// TwinCAT 3 PLC project Clara_20230419
// ProgramVersion: 3.1.4022.7
// CompilerDefines: VISU_USEWSTRING
// libraries:
//   CAA Memory, * (CAA Technical Workgroup)
//   CmpBitmapPool, * (System)
//   Tc2_EtherCAT, * (Beckhoff Automation GmbH)
//   Tc2_IoFunctions, * (Beckhoff Automation GmbH)
//   Tc2_MC2, * (Beckhoff Automation GmbH)
//   Tc2_MDP, * (Beckhoff Automation GmbH)
//   Tc2_ModbusRTU, * (Beckhoff Automation GmbH)
//   Tc2_SerialCom, * (Beckhoff Automation GmbH)
//   Tc2_Standard, * (Beckhoff Automation GmbH)
//   Tc2_SUPS, * (Beckhoff Automation GmbH)
//   Tc2_System, * (Beckhoff Automation GmbH)
//   Tc2_SystemCX, * (Beckhoff Automation GmbH)
//   Tc2_Utilities, * (Beckhoff Automation GmbH)
//   Tc3_Module, * (Beckhoff Automation GmbH)
//   VisuDialogs, * (System)
//   VisuSymbols,3.5.10.0,System
// project tree:
//   DUTs/01_ST_IO/ ST_Input.TcDUT, ST_IO_FootPedal.TcDUT, ST_Output.TcDUT (not stored)
//   DUTs/02_PLC/ stAxis.TcDUT, stFootPedal.TcDUT (not stored), stISS.TcDUT, stSubTank.TcDUT, stMaintenanceUnit.TcDUT (not stored), stRollToRoll.TcDUT (not stored), stRtu.TcDUT, stSafetyGuard.TcDUT (not stored), stSpitUnit.TcDUT, stSystemEnvironment.TcDUT (not stored), stTableVacuum.TcDUT, stUpDownSlot.TcDUT (not stored), stUVLed.TcDUT
//   Enum_Text/Enum/PLC/ AxisStateEnum.TcDUT, Axis_XY_ErrorEnum.TcDUT, Axis_Z_ErrorEnum.TcDUT (not stored), EnvironmentErrorEnum.TcDUT (not stored), EnvironmentStateEnum.TcDUT (not stored), FootPedalErrorEnum.TcDUT, FootPedalStateEnum.TcDUT, ISSErrorEnum.TcDUT, SubTankErrorEnum.TcDUT (not stored), ISSStateEnum.TcDUT (not stored), SubTankInkEnum.TcDUT, SubTankStateEnum.TcDUT, MUErrorEnum.TcDUT, MUStateEnum.TcDUT, RTRErrorEnum.TcDUT (not stored), RTRStateEnum.TcDUT (not stored), SafetyGuardErrorEnum.TcDUT (not stored), SafetyGuardStateEnum.TcDUT (not stored), SpitUnitErrorEnum.TcDUT (not stored), SpitUnitStateEnum.TcDUT (not stored), SwapInfoEnum.TcDUT, TabVacErrorEnum.TcDUT (not stored), TabVacStateEnum.TcDUT, UpDownSlotErrorEnum.TcDUT (not stored), UpDownSlotStateEnum.TcDUT (not stored), UVLedErrorEnum.TcDUT (not stored), UVLedStateEnum.TcDUT (not stored)
//   Enum_Text/Enum/TwinSafe/ TwinSAFE_FB_ESTOP_State_Enum.TcDUT, TwinSAFE_Group_State_Enum.TcDUT (not stored)
//   Global Variables/ _01_Global_Variables.TcGVL, _04_Global_Variables_InOutput.TcGVL
//   / GlobalTextList.TcGTLO, ImagePool.TcIPO (not stored), PlcTask.TcTTO, Task_com.TcTTO, 视图管理器.TcVMO (not stored)
//   GVLs/ COMM.TcGVL, GVL.TcGVL, GVL_Alarm.TcGVL, GVL_API.TcGVL (not stored)
//   POUs/000_程序辅助系统/报警/Data types/ Alm_AlarmHistoryType.TcDUT (not stored), Alm_AlarmType.TcDUT, Alm_AlmMsg.TcDUT, Alm_EventClass.TcDUT
//   POUs/000_程序辅助系统/报警/diag_FB/ ethercatinfo_read.TcPOU (not stored)
//   POUs/000_程序辅助系统/报警/Alarm_FB/ FB_AlarmMain.TcPOU, FB_DiagDataLogging_S.TcPOU (not stored), FB_SetAlarm.TcPOU (not stored), SW_FormatWstring.TcPOU
//   POUs/000_程序辅助系统/报警/Alarm_FB/Products/ FB_DirectoryCopy.TcPOU (not stored), FB_FileCopy.TcPOU
//   POUs/000_程序辅助系统/报警/ MAIN_Alarm.TcPOU (not stored)
//   POUs/000_程序辅助系统/系统功能/ P_UPS.TcPOU (not stored), systime.TcPOU
//   POUs/001_FB/ FB_Buzzer.TcPOU, FB_count.TcPOU (not stored), FB_SQUARE.TcPOU, FB_WriteAnalog.TcPOU (not stored)
//   POUs/002_Modbus/BackPrg/ PRG_COMM.TcPOU
//   POUs/002_Modbus/ PRG_SerialComm.TcPOU (not stored), P_Modbus.TcPOU, P_Modbus_RTU.TcPOU (not stored)
//   POUs/003_Input_Output/ IO_Link.TcPOU, P_API_IO.TcPOU (not stored)
//   POUs/010_Motion/MotionBase/ FB_Home_Z.TcPOU (not stored), FB_Home_X.TcPOU, FB_MoveFS_Exte.TcPOU, FB_MoveSS_Exte.TcPOU, FB_MoveZ_Exte.TcPOU
//   POUs/010_Motion/XMove/ P_FastScan.TcPOU
//   POUs/010_Motion/YMove/ P_SlowScan.TcPOU
//   POUs/010_Motion/ZMove/ P_Z_Axis.TcPOU
//   POUs/030_MediaTransport/TableVacuum/FB/ FB_TableVacuum.TcPOU (not stored)
//   POUs/030_MediaTransport/UpDownSlot/FB/ FB_UpDownSlotS1.TcPOU, FB_UpDownSlotS2_S6.TcPOU
//   POUs/040_System/FootPedal/FB/ FB_FootPedal.TcPOU
//   POUs/040_System/SafetyGuard/FB/ FB_SafetyGuard.TcPOU (not stored)
//   POUs/040_System/SafetyGuard/ P_SafetyGuard.TcPOU (not stored)
//   POUs/040_System/SystemEnvironment/FB/ FB_SystemEnvironment.TcPOU
//   POUs/050_InkSystem/ISS/ P_ISS.TcPOU
//   POUs/050_InkSystem/ P_InkSystem.TcPOU (not stored)
//   POUs/050_InkSystem/搅拌_吸废墨/FB/ FB_Stirrer.TcPOU (not stored)
//   POUs/050_InkSystem/搅拌_吸废墨/ P_Stirrer_WastePump.TcPOU (not stored)
//   POUs/030_MediaTransport/ P_MediaTransport.TcPOU
//   POUs/030_MediaTransport/TableVacuum/ P_TableVacuum.TcPOU (not stored)
//   POUs/030_MediaTransport/UpDownSlot/ P_UpDownSlot.TcPOU (not stored)
//   POUs/010_Motion/MotionBase/PTP/ Axis_IO.TcPOU, Axis_PTP_CoE.TcPOU (not stored)
//   POUs/010_Motion/ P_Motion.TcPOU (not stored)
//   POUs/060_UVLed/FB/ FB_UVLed_L.TcPOU (not stored), FB_UVLed_R.TcPOU (not stored)
//   POUs/070_RollToRoll/FB/ FB_RollToRoll_Torque.TcPOU
//   POUs/100_SubTank/FB/ FB_Circulation.TcPOU, FB_SubTank_C.TcPOU, FB_SubTank_W.TcPOU
//   POUs/100_SubTank/ P_SubTank.TcPOU
//   POUs/999_TwinSAFE/ P_TwinSAFE.TcPOU
//   POUs/ MAIN.TcPOU (not stored)
//   POUs/070_RollToRoll/ P_RollToRoll.TcPOU (not stored)
//   POUs/040_System/FootPedal/ P_FootPedal.TcPOU (not stored)
//   POUs/040_System/ P_System.TcPOU (not stored)
//   POUs/040_System/SystemEnvironment/ P_SystemEnvironment.TcPOU
//   POUs/060_UVLed/ P_UVLed.TcPOU (not stored)
//   POUs/090MaintenanceUnit/FB/ FB_Auto_Cycles_Swap.TcPOU (not stored), FB_drip_purge.TcPOU
//   POUs/090MaintenanceUnit/ P_MaintenanceUnit.TcPOU (not stored)
//   POUs/080SpitUnit/FB/ FB_HomeSpitUnit.TcPOU, FB_MoveSpitUnit_Exte.TcPOU
//   POUs/080SpitUnit/ P_SpitUnit.TcPOU
//   VISUs/base/ title.TcVIS
//   VISUs/Components/IO_Components/ F99_IO_IO.TcVIS, F99_IO_IO_1.TcVIS, F99_IO_IO_2.TcVIS
//   VISUs/Components/ VIS_FootPedal.TcVIS (not stored), VIS_Drip_purge.TcVIS (not stored), VIS_SubTank.TcVIS, VIS_SystemEnvironment.TcVIS (not stored), VIS_ISS.TcVIS (not stored), VIS_MU.TcVIS (not stored), VIS_RTR_1.TcVIS (not stored), VIS_RTR_2.TcVIS, VIS_SaftyGuard.TcVIS (not stored), VIS_SpitUnit.TcVIS, VIS_TabVac.TcVIS, VIS_UpDownSlot.TcVIS
//   VISUs/HMI_IO监控文字/ EL1809_M_1.TcTLO, EL1809_M_2.TcTLO, EL1809_M_3.TcTLO, EL1809_S_1.TcTLO, EL1809_S_2.TcTLO (not stored), EL1904_M_1.TcTLO, EL1904_M_2.TcTLO, EL1904_M_3.TcTLO (not stored), EL1904_M_4.TcTLO (not stored), EL1904_M_5.TcTLO (not stored), EL2809_M_1.TcTLO (not stored), EL2809_M_2.TcTLO (not stored), EL2809_M_3.TcTLO (not stored), EL2809_M_4.TcTLO, EL2809_S_1.TcTLO (not stored), EL2904_M_1.TcTLO (not stored)
//   VISUs/ F99_Monitor.TcVIS (not stored), F7_RTR.TcVIS, F4_System.TcVIS (not stored), F1_AXIS.TcVIS, F5_InkSystem.TcVIS, F3_MediaTransport.TcVIS (not stored), F6_UVLed.TcVIS (not stored)
//   VISUs/VIS文本/PLC/ ISS_Object.TcTLO, subinklevel.TcTLO (not stored), TextListSpitUnitErrorid.TcTLO (not stored), TextListSpitUnitState.TcTLO, TextList_EnvironmentError.TcTLO, TextList_EnvironmentState.TcTLO, TextList_FootPedalerroid.TcTLO (not stored), TextList_SubTankerroid.TcTLO, TextList_FootPedalstate.TcTLO, TextList_ISSerrorid.TcTLO, TextList_ISSstate.TcTLO, TextList_MU_errorid.TcTLO, TextList_MU_state.TcTLO, TextList_RTRstate.TcTLO (not stored), TextList_RTR_errorid.TcTLO, TextList_SafetyGuarderrorid.TcTLO (not stored), TextList_SafetyGuardstate.TcTLO, TextList_SubTank_circuit.TcTLO, TextList_SwapInfo.TcTLO, TextList_tabvac_errorid.TcTLO, TextList_tabvac_state.TcTLO, TextList_UpDownSlot_errorid.TcTLO, TextList_UpDownSlot_state.TcTLO, TextList_UVLed_errorid.TcTLO (not stored), TextList_UVLed_state.TcTLO (not stored), TextList_xyErrorid.TcTLO, TextList_xyzState.TcTLO, TextList_zErrorid.TcTLO (not stored)
//   VISUs/VIS文本/TwinSafe/ TextList_TwinSAFE_FB_ESTOP_State.TcTLO, TextList_TwinSAFE_Group_State.TcTLO
//   VISUs/报警/ Visualization_ActEvent.TcVIS, Visualization_LogEvent.TcVIS (not stored), vis_arm.TcVIS
// real-time tasks:
//   TASK PlcTask: cycle T#10ms, priority 12, ADS port 350
//   TASK Task_com: cycle T#2ms, priority 6, ADS port 352
// motion (NC):
//   TASK NC-Task 1 SAF: cycle T#2ms, priority 4, ADS port 501
//   TASK NC-Task 1 SVB: cycle T#5ms, priority 10, ADS port 511
//   AXIS Axis_FS (id 1)
//     Dynamic: Acceleration=5927.27, Deceleration=5927.27, Jerk=27883
//     Velo: RefSearch=10, RefSync=10, SlowManual=50, FastManual=100
//     TargetPosControl: Time=0.005
//     OtherSettings: AllowMotionCmdToSlave=true
//     encoder EncType=19
//       EncPara: ScaleFactorNumerator=0.001, MaxCount=#xffffffff
//         Inc: RefSearchInverse=true, RefSyncInverse=false
//     drive DrvType=16
//       DrvPara: MaxCount=#xffffffff, DriveControlDWord=#x00020000
//         Analog: VeloReferenz=2000, TorqueSetpointScale=10, ScaleFactorActTorque=0.1
//         TimeComp: TaskDelayCycles=1
//     controller CtrType=1
//       CtrPara: PriorControlFactor=1
//         PosDiffControl: Range=250
//         Observer: BandWidth=20
//   AXIS Axis_SS (id 2)
//     Dynamic: Acceleration=274.92, Deceleration=274.92, Jerk=748.92
//     Velo: Maximum=174
//     OtherSettings: AllowMotionCmdToSlave=true
//     encoder EncType=19
//       EncPara: ScaleFactorNumerator=3.12605035e-07, Inverse=true, MaxCount=#xffffffff
//     drive DrvType=16
//       DrvPara: Inverse=true, MaxCount=#xffffffff, DriveControlDWord=#x00020000
//         Analog: VeloReferenz=180, TorqueSetpointScale=10, ScaleFactorActTorque=0.1
//         TimeComp: TaskDelayCycles=1
//     controller CtrType=1
//       CtrPara: PriorControlFactor=1
//         PosDiffControl: Range=50
//         Observer: BandWidth=20
//   AXIS Z_Axis (id 3)
//     Dynamic: Acceleration=33.4286, Deceleration=33.4286, Jerk=133.032
//     Velo: RefSearch=2, RefSync=2, SlowManual=8, FastManual=10, Maximum=15
//     OtherSettings: AllowMotionCmdToSlave=true
//     encoder EncType=19
//       EncPara: ScaleFactorNumerator=1.7881393e-08, MaxCount=#xffffffff
//         Inc: RefSearchInverse=true, RefSyncInverse=false
//     drive DrvType=16
//       DrvPara: MaxCount=#xffffffff, DriveControlDWord=#x00020000
//         Analog: VeloReferenz=15, TorqueSetpointScale=10, ScaleFactorActTorque=0.1
//         TimeComp: TaskDelayCycles=1
//     controller CtrType=1
//       CtrPara: PriorControlFactor=1
//         PosDiffControl: Range=10
//         Observer: BandWidth=20
//   AXIS Axis_unwider_input1 (id 4)
//     Dynamic: Acceleration=4200, Deceleration=4200, Jerk=14700
//     Velo: SlowManual=60, FastManual=100, Maximum=3000
//     OtherSettings: AllowMotionCmdToSlave=true
//     encoder EncType=19
//       EncPara: ScaleFactorNumerator=3.57628e-06, MaxCount=#xffffffff
//     drive DrvType=16
//       DrvPara: MaxCount=#xffffffff, DriveControlDWord=#x00020000
//         Analog: VeloReferenz=3000, TorqueSetpointScale=10, ScaleFactorActTorque=0.1
//         TimeComp: TaskDelayCycles=1
//     controller CtrType=1
//       CtrPara: PriorControlFactor=1
//         PosDiffControl: Enable=false, Range=100
//         Observer: BandWidth=20
//   AXIS Axis_unwinder_input2 (id 5)
//     Dynamic: Acceleration=4000, Deceleration=4000, Jerk=16000
//     Velo: Maximum=3000
//     OtherSettings: AllowMotionCmdToSlave=true
//     encoder EncType=19
//       EncPara: ScaleFactorNumerator=3.57628e-06, Inverse=true, MaxCount=#xffffffff
//     drive DrvType=16
//       DrvPara: Inverse=true, MaxCount=#xffffffff, DriveControlDWord=#x00020000
//         Analog: VeloReferenz=3000, TorqueSetpointScale=10, ScaleFactorActTorque=0.1
//         TimeComp: TaskDelayCycles=1
//     controller CtrType=1
//       CtrPara: PriorControlFactor=1
//         PosDiffControl: Enable=false, Range=100
//         Observer: BandWidth=20
//   AXIS Axis_winder_output1 (id 6)
//     Dynamic: Acceleration=4000, Deceleration=4000, Jerk=16000
//     Velo: Maximum=3000
//     OtherSettings: AllowMotionCmdToSlave=true
//     encoder EncType=19
//       EncPara: ScaleFactorNumerator=3.57628e-06, MaxCount=#xffffffff
//     drive DrvType=16
//       DrvPara: MaxCount=#xffffffff, DriveControlDWord=#x00020000
//         Analog: VeloReferenz=3000, TorqueSetpointScale=10, ScaleFactorActTorque=0.1
//         TimeComp: TaskDelayCycles=1
//     controller CtrType=1
//       CtrPara: PriorControlFactor=1
//         PosDiffControl: Enable=false, Range=100
//         Observer: BandWidth=20
//   AXIS Axis_winder_output2 (id 7)
//     Dynamic: Acceleration=4000, Deceleration=4000, Jerk=16000
//     Velo: Maximum=3000
//     OtherSettings: AllowMotionCmdToSlave=true
//     encoder EncType=19
//       EncPara: ScaleFactorNumerator=3.57628e-06, Inverse=true, MaxCount=#xffffffff
//     drive DrvType=16
//       DrvPara: Inverse=true, MaxCount=#xffffffff, DriveControlDWord=#x00020000
//         Analog: VeloReferenz=3000, TorqueSetpointScale=10, ScaleFactorActTorque=0.1
//         TimeComp: TaskDelayCycles=1
//     controller CtrType=1
//       CtrPara: PriorControlFactor=1
//         PosDiffControl: Enable=false, Range=100
//         Observer: BandWidth=20
//   AXIS SpitUnit (id 8)
//     Dynamic: Acceleration=32.1429, Deceleration=32.1429, Jerk=137.755
//     Velo: RefSearch=2, RefSync=2, SlowManual=5, FastManual=10, Maximum=15
//     OtherSettings: AllowMotionCmdToSlave=true
//     encoder EncType=19
//       EncPara: ScaleFactorNumerator=1.7881393e-08, Inverse=true, MaxCount=#xffffffff
//         Inc: RefSearchInverse=true, RefSyncInverse=false
//     drive DrvType=16
//       DrvPara: Inverse=true, MaxCount=#xffffffff, DriveControlDWord=#x00020000
//         Analog: VeloReferenz=15, TorqueSetpointScale=10, ScaleFactorActTorque=0.1
//         TimeComp: TaskDelayCycles=1
//     controller CtrType=1
//       CtrPara: PriorControlFactor=1
//         PosDiffControl: Range=10
//         Observer: BandWidth=20
// I/O:
//   DEVICE Device 1 (EtherCAT), AmsNetId 192.168.1.138.2.1
//     Term 1 (EK1200) [EK1200-5000 EtherCAT Power supply (2A E-Bus)]
//       Term 2 (EL1809) [EL1809 16Ch. Dig. Input 24V, 3ms]
//       Term 3 (EL1809) [EL1809 16Ch. Dig. Input 24V, 3ms]
//       Term 4 (EL1809) [EL1809 16Ch. Dig. Input 24V, 3ms]
//       Term 5 (EL2809) [EL2809 16Ch. Dig. Output 24V, 0.5A]
//       Term 6 (EL2809) [EL2809 16Ch. Dig. Output 24V, 0.5A]
//       Term 7 (EL2809) [EL2809 16Ch. Dig. Output 24V, 0.5A]
//       Term 8 (EL6900) [EL6900, TwinSAFE PLC]
//       Term 9 (EL1904) [EL1904, 4 Ch. Safety Input 24V, TwinSAFE]
//         modules: Module 1 (FSOES)
//       Term 10 (EL1904) [EL1904, 4 Ch. Safety Input 24V, TwinSAFE]
//         modules: Module 1 (FSOES)
//       Term 11 (EL1904) [EL1904, 4 Ch. Safety Input 24V, TwinSAFE]
//         modules: Module 1 (FSOES)
//       Term 12 (EL1904) [EL1904, 4 Ch. Safety Input 24V, TwinSAFE]
//         modules: Module 1 (FSOES)
//       Term 13 (EL1904) [EL1904, 4 Ch. Safety Input 24V, TwinSAFE]
//         modules: Module 1 (FSOES)
//       Term 14 (EL9410) [EL9410 E-Bus Power Supplier  (Diagnostics)]
//       Term 15 (EL2904) [EL2904, 4 Ch. Safety Output 24V, 0.5A, TwinSAFE]
//         modules: Module 1 (FSOES), Module 2 (DO)
//       Term 16 (EL2809) [EL2809 16Ch. Dig. Output 24V, 0.5A]
//       Term 17 (EL6001) [EL6001 Interface (RS232)]
//       Term 18 (EL6022) [EL6022 Interface 2Ch. (RS422/485)]
//       Term 19 (EK1110) [EK1110 EtherCAT extension]
//     Drive 20 (ASDA-A3-E CoE Drive) [Delta ASDA-A3-E EtherCAT(CoE) Drive Rev0.05]
//     Drive 21 (ASDA-A3-E CoE Drive) [Delta ASDA-A3-E EtherCAT(CoE) Drive Rev0.05]
//     Drive 22 (ASDA-A3-E CoE Drive) [Delta ASDA-A3-E EtherCAT(CoE) Drive Rev0.05]
//     Drive 23 (ASDA-A3-E CoE Drive) [Delta ASDA-A3-E EtherCAT(CoE) Drive Rev0.05]
//     Drive 24 (ASDA-A3-E CoE Drive) [Delta ASDA-A3-E EtherCAT(CoE) Drive Rev0.05]
//     Drive 25 (ASDA-A3-E CoE Drive) [Delta ASDA-A3-E EtherCAT(CoE) Drive Rev0.05]
//     Drive 26 (ASDA-A3-E CoE Drive) [Delta ASDA-A3-E EtherCAT(CoE) Drive Rev0.05]
//     Drive 27 (ASDA-A3-E CoE Drive) [Delta ASDA-A3-E EtherCAT(CoE) Drive Rev0.05]
//     Term 28 (EK1100) [EK1100 EtherCAT Coupler (2A E-Bus)]
//       Term 29 (EL1809) [EL1809 16Ch. Dig. Input 24V, 3ms]
//       Term 30 (EL1809) [EL1809 16Ch. Dig. Input 24V, 3ms]
//       Term 31 (EL2809) [EL2809 16Ch. Dig. Output 24V, 0.5A]
//       Term 32 (EL4002) [EL4002 2Ch. Ana. Output 0-10V, 12bit]
//       Term 33 (EL9011) [EL9011 End Terminal]
// variable links:
//   Device 1 (EtherCAT) <-> Device 1 (EtherCAT)/Term 1 (EK1200)/Term 10 (EL1904)
//     Term 1 (EK1200)/Term 8 (EL6900)/ConnectionInputs/Message_53 TxPDO <-> Module 1 (FSOES)/RxPDO/FSOE
//   Device 1 (EtherCAT) <-> Device 1 (EtherCAT)/Term 1 (EK1200)/Term 12 (EL1904)
//     Term 1 (EK1200)/Term 8 (EL6900)/ConnectionOutputs/Message_55 RxPDO <-> Module 1 (FSOES)/TxPDO/FSOE
//   Device 1 (EtherCAT) <-> Device 1 (EtherCAT)/Term 1 (EK1200)/Term 13 (EL1904)
//     Term 1 (EK1200)/Term 8 (EL6900)/ConnectionInputs/Message_56 TxPDO <-> Module 1 (FSOES)/RxPDO/FSOE
//     Term 1 (EK1200)/Term 8 (EL6900)/ConnectionOutputs/Message_56 RxPDO <-> Module 1 (FSOES)/TxPDO/FSOE
//   Device 1 (EtherCAT) <-> Device 1 (EtherCAT)/Term 1 (EK1200)/Term 15 (EL2904)
//     Term 1 (EK1200)/Term 8 (EL6900)/ConnectionInputs/Message_57 TxPDO <-> Module 1 (FSOES)/RxPDO/FSOE
//   Device 1 (EtherCAT) <-> Device 1 (EtherCAT)/Term 1 (EK1200)/Term 8 (EL6900)
//     Term 1 (EK1200)/Term 10 (EL1904)/Module 1 (FSOES)/TxPDO/FSOE <-> ConnectionOutputs/Message_53 RxPDO
//     Term 1 (EK1200)/Term 11 (EL1904)/Module 1 (FSOES)/TxPDO/FSOE <-> ConnectionOutputs/Message_58 RxPDO
//     Term 1 (EK1200)/Term 15 (EL2904)/Module 1 (FSOES)/TxPDO/FSOE <-> ConnectionOutputs/Message_57 RxPDO
//     Term 1 (EK1200)/Term 11 (EL1904)/Module 1 (FSOES)/RxPDO/FSOE <-> ConnectionInputs/Message_58 TxPDO
//     Term 1 (EK1200)/Term 12 (EL1904)/Module 1 (FSOES)/RxPDO/FSOE <-> ConnectionInputs/Message_55 TxPDO
//     Term 1 (EK1200)/Term 9 (EL1904)/Module 1 (FSOES)/RxPDO/FSOE <-> ConnectionInputs/Message_52 TxPDO
//   Device 1 (EtherCAT) <-> Device 1 (EtherCAT)/Term 1 (EK1200)/Term 9 (EL1904)
//     Term 1 (EK1200)/Term 8 (EL6900)/ConnectionOutputs/Message_52 RxPDO <-> Module 1 (FSOES)/TxPDO/FSOE
//   NC-Task 1 SAF/Axes/Axis_FS <-> Device 1 (EtherCAT)/Drive 20 (ASDA-A3-E CoE Drive)
//     Drive/Inputs/In/nDataIn3[0] <-> 2nd TxPDO Mapping/Actual Torque
//     Drive/Inputs/In/nDcOutputTime <-> InfoData/DcOutputShift
//     Drive/Inputs/In/nState1 <-> 2nd TxPDO Mapping/Status Word
//     Drive/Inputs/In/nState2 <-> 2nd TxPDO Mapping/Status Word @bit 8
//     Drive/Inputs/In/nState4 @bit 1 <-> WcState/InputToggle
//     Drive/Inputs/In/nState4 <-> WcState/WcState
//     Drive/Outputs/Out/nCtrl1 <-> 2nd RxPDO Mapping/Control Word
//     Drive/Outputs/Out/nCtrl2 <-> 2nd RxPDO Mapping/Control Word @bit 8
//     Drive/Outputs/Out/nDataOut1 <-> 2nd RxPDO Mapping/Target Position
//     Drive/Outputs/Out/nDataOut2 <-> 2nd RxPDO Mapping/Target Velocity
//     Drive/Outputs/Out/nDataOut4[0] <-> 2nd RxPDO Mapping/Target Torque
//     Enc/Inputs/In/nDataIn1 <-> 2nd TxPDO Mapping/Actual Position
//     Enc/Inputs/In/nDataIn3 <-> 2nd TxPDO Mapping/Touch Probe Pos1 Pos Value
//     Enc/Inputs/In/nDataIn7 <-> 2nd TxPDO Mapping/Velocity actual value
//     Enc/Inputs/In/nDcInputTime <-> InfoData/DcInputShift
//     Enc/Inputs/In/nState4 @bit 1 <-> WcState/InputToggle
//     Enc/Inputs/In/nState4 <-> WcState/WcState
//     Enc/Inputs/In/nState5 <-> 2nd TxPDO Mapping/Touch Probe Status
//     Enc/Inputs/In/nState6 <-> 2nd TxPDO Mapping/Touch Probe Status @bit 8
//     Enc/Outputs/Out/nCtrl5 <-> 2nd RxPDO Mapping/Touch Probe Function
//     Enc/Outputs/Out/nCtrl6 <-> 2nd RxPDO Mapping/Touch Probe Function @bit 8
//   NC-Task 1 SAF/Axes/Axis_SS <-> Device 1 (EtherCAT)/Drive 21 (ASDA-A3-E CoE Drive)
//     Drive/Inputs/In/nDataIn3[0] <-> 2nd TxPDO Mapping/Actual Torque
//     Drive/Inputs/In/nDcOutputTime <-> InfoData/DcOutputShift
//     Drive/Inputs/In/nState1 <-> 2nd TxPDO Mapping/Status Word
//     Drive/Inputs/In/nState2 <-> 2nd TxPDO Mapping/Status Word @bit 8
//     Drive/Inputs/In/nState4 @bit 1 <-> WcState/InputToggle
//     Drive/Inputs/In/nState4 <-> WcState/WcState
//     Drive/Outputs/Out/nCtrl1 <-> 2nd RxPDO Mapping/Control Word
//     Drive/Outputs/Out/nCtrl2 <-> 2nd RxPDO Mapping/Control Word @bit 8
//     Drive/Outputs/Out/nDataOut1 <-> 2nd RxPDO Mapping/Target Position
//     Drive/Outputs/Out/nDataOut2 <-> 2nd RxPDO Mapping/Target Velocity
//     Drive/Outputs/Out/nDataOut4[0] <-> 2nd RxPDO Mapping/Target Torque
//     Enc/Inputs/In/nDataIn1 <-> 2nd TxPDO Mapping/Actual Position
//     Enc/Inputs/In/nDataIn3 <-> 2nd TxPDO Mapping/Touch Probe Pos1 Pos Value
//     Enc/Inputs/In/nDataIn7 <-> 2nd TxPDO Mapping/Velocity actual value
//     Enc/Inputs/In/nDcInputTime <-> InfoData/DcInputShift
//     Enc/Inputs/In/nState4 @bit 1 <-> WcState/InputToggle
//     Enc/Inputs/In/nState4 <-> WcState/WcState
//     Enc/Inputs/In/nState5 <-> 2nd TxPDO Mapping/Touch Probe Status
//     Enc/Inputs/In/nState6 <-> 2nd TxPDO Mapping/Touch Probe Status @bit 8
//     Enc/Outputs/Out/nCtrl5 <-> 2nd RxPDO Mapping/Touch Probe Function
//     Enc/Outputs/Out/nCtrl6 <-> 2nd RxPDO Mapping/Touch Probe Function @bit 8
//   NC-Task 1 SAF/Axes/Axis_unwider_input1 <-> Device 1 (EtherCAT)/Drive 23 (ASDA-A3-E CoE Drive)
//     Drive/Inputs/In/nDataIn3[0] <-> 3rd TxPDO Mapping/Actual Torque
//     Drive/Inputs/In/nDcOutputTime <-> InfoData/DcOutputShift
//     Drive/Inputs/In/nState1 <-> 3rd TxPDO Mapping/Status Word
//     Drive/Inputs/In/nState2 <-> 3rd TxPDO Mapping/Status Word @bit 8
//     Drive/Inputs/In/nState4 @bit 1 <-> WcState/InputToggle
//     Drive/Inputs/In/nState4 <-> WcState/WcState
//     Drive/Inputs/In/nState5 <-> 3rd TxPDO Mapping/Mode Of Operation Display
//     Drive/Outputs/Out/nCtrl1 <-> 3rd RxPDO Mapping/Control Word
//     Drive/Outputs/Out/nCtrl2 <-> 3rd RxPDO Mapping/Control Word @bit 8
//     Drive/Outputs/Out/nCtrl5 <-> 3rd RxPDO Mapping/Mode Of Operation
//     Drive/Outputs/Out/nDataOut1 <-> 3rd RxPDO Mapping/Target Position
//     Drive/Outputs/Out/nDataOut2 <-> 3rd RxPDO Mapping/Target Velocity
//     Drive/Outputs/Out/nDataOut4[0] <-> 3rd RxPDO Mapping/Target Torque
//     Enc/Inputs/In/nDataIn1 <-> 3rd TxPDO Mapping/Actual Position
//     Enc/Inputs/In/nDataIn3 <-> 3rd TxPDO Mapping/Touch Probe Pos1 Pos Value
//     Enc/Inputs/In/nDataIn7 <-> 3rd TxPDO Mapping/Velocity actual value
//     Enc/Inputs/In/nDcInputTime <-> InfoData/DcInputShift
//     Enc/Inputs/In/nState4 @bit 1 <-> WcState/InputToggle
//     Enc/Inputs/In/nState4 <-> WcState/WcState
//     Enc/Inputs/In/nState5 <-> 3rd TxPDO Mapping/Touch Probe Status
//     Enc/Inputs/In/nState6 <-> 3rd TxPDO Mapping/Touch Probe Status @bit 8
//     Enc/Outputs/Out/nCtrl5 <-> 3rd RxPDO Mapping/Touch Probe Function
//     Enc/Outputs/Out/nCtrl6 <-> 3rd RxPDO Mapping/Touch Probe Function @bit 8
//   NC-Task 1 SAF/Axes/Axis_unwinder_input2 <-> Device 1 (EtherCAT)/Drive 24 (ASDA-A3-E CoE Drive)
//     Drive/Inputs/In/nDataIn3[0] <-> 3rd TxPDO Mapping/Actual Torque
//     Drive/Inputs/In/nDcOutputTime <-> InfoData/DcOutputShift
//     Drive/Inputs/In/nState1 <-> 3rd TxPDO Mapping/Status Word
//     Drive/Inputs/In/nState2 <-> 3rd TxPDO Mapping/Status Word @bit 8
//     Drive/Inputs/In/nState4 @bit 1 <-> WcState/InputToggle
//     Drive/Inputs/In/nState4 <-> WcState/WcState
//     Drive/Inputs/In/nState5 <-> 3rd TxPDO Mapping/Mode Of Operation Display
//     Drive/Outputs/Out/nCtrl1 <-> 3rd RxPDO Mapping/Control Word
//     Drive/Outputs/Out/nCtrl2 <-> 3rd RxPDO Mapping/Control Word @bit 8
//     Drive/Outputs/Out/nCtrl5 <-> 3rd RxPDO Mapping/Mode Of Operation
//     Drive/Outputs/Out/nDataOut1 <-> 3rd RxPDO Mapping/Target Position
//     Drive/Outputs/Out/nDataOut2 <-> 3rd RxPDO Mapping/Target Velocity
//     Drive/Outputs/Out/nDataOut4[0] <-> 3rd RxPDO Mapping/Target Torque
//     Enc/Inputs/In/nDataIn1 <-> 3rd TxPDO Mapping/Actual Position
//     Enc/Inputs/In/nDataIn3 <-> 3rd TxPDO Mapping/Touch Probe Pos1 Pos Value
//     Enc/Inputs/In/nDataIn7 <-> 3rd TxPDO Mapping/Velocity actual value
//     Enc/Inputs/In/nDcInputTime <-> InfoData/DcInputShift
//     Enc/Inputs/In/nState4 @bit 1 <-> WcState/InputToggle
//     Enc/Inputs/In/nState4 <-> WcState/WcState
//     Enc/Inputs/In/nState5 <-> 3rd TxPDO Mapping/Touch Probe Status
//     Enc/Inputs/In/nState6 <-> 3rd TxPDO Mapping/Touch Probe Status @bit 8
//     Enc/Outputs/Out/nCtrl5 <-> 3rd RxPDO Mapping/Touch Probe Function
//     Enc/Outputs/Out/nCtrl6 <-> 3rd RxPDO Mapping/Touch Probe Function @bit 8
//   NC-Task 1 SAF/Axes/Axis_winder_output1 <-> Device 1 (EtherCAT)/Drive 25 (ASDA-A3-E CoE Drive)
//     Drive/Inputs/In/nDataIn3[0] <-> 3rd Transmit PDO Mapping/Torque actual value
//     Drive/Inputs/In/nDcOutputTime <-> InfoData/DcOutputShift
//     Drive/Inputs/In/nState1 <-> 3rd Transmit PDO Mapping/Statusword
//     Drive/Inputs/In/nState2 <-> 3rd Transmit PDO Mapping/Statusword @bit 8
//     Drive/Inputs/In/nState4 @bit 1 <-> WcState/InputToggle
//     Drive/Inputs/In/nState4 <-> WcState/WcState
//     Drive/Inputs/In/nState5 <-> 3rd Transmit PDO Mapping/Modes of operation display
//     Drive/Outputs/Out/nCtrl1 <-> 3rd Receive PDO Mapping/Controlword
//     Drive/Outputs/Out/nCtrl2 <-> 3rd Receive PDO Mapping/Controlword @bit 8
//     Drive/Outputs/Out/nCtrl5 <-> 3rd Receive PDO Mapping/Modes of operation
//     Drive/Outputs/Out/nDataOut1 <-> 3rd Receive PDO Mapping/Target position
//     Drive/Outputs/Out/nDataOut2 <-> 3rd Receive PDO Mapping/Target velocity
//     Drive/Outputs/Out/nDataOut4[0] <-> 3rd Receive PDO Mapping/Target torque
//     Enc/Inputs/In/nDataIn1 <-> 3rd Transmit PDO Mapping/Position actual value
//     Enc/Inputs/In/nDataIn3 <-> 3rd Transmit PDO Mapping/Touch Probe Pos1 Pos Value
//     Enc/Inputs/In/nDataIn7 <-> 3rd Transmit PDO Mapping/Velocity actual value
//     Enc/Inputs/In/nDcInputTime <-> InfoData/DcInputShift
//     Enc/Inputs/In/nState4 @bit 1 <-> WcState/InputToggle
//     Enc/Inputs/In/nState4 <-> WcState/WcState
//     Enc/Inputs/In/nState5 <-> 3rd Transmit PDO Mapping/Touch Probe Status
//     Enc/Inputs/In/nState6 <-> 3rd Transmit PDO Mapping/Touch Probe Status @bit 8
//     Enc/Outputs/Out/nCtrl5 <-> 3rd Receive PDO Mapping/Touch Probe Function
//     Enc/Outputs/Out/nCtrl6 <-> 3rd Receive PDO Mapping/Touch Probe Function @bit 8
//   NC-Task 1 SAF/Axes/Axis_winder_output2 <-> Device 1 (EtherCAT)/Drive 26 (ASDA-A3-E CoE Drive)
//     Drive/Inputs/In/nDataIn3[0] <-> 3rd TxPDO Mapping/Actual Torque
//     Drive/Inputs/In/nDcOutputTime <-> InfoData/DcOutputShift
//     Drive/Inputs/In/nState1 <-> 3rd TxPDO Mapping/Status Word
//     Drive/Inputs/In/nState2 <-> 3rd TxPDO Mapping/Status Word @bit 8
//     Drive/Inputs/In/nState4 @bit 1 <-> WcState/InputToggle
//     Drive/Inputs/In/nState4 <-> WcState/WcState
//     Drive/Inputs/In/nState5 <-> 3rd TxPDO Mapping/Mode Of Operation Display
//     Drive/Outputs/Out/nCtrl1 <-> 3rd RxPDO Mapping/Control Word
//     Drive/Outputs/Out/nCtrl2 <-> 3rd RxPDO Mapping/Control Word @bit 8
//     Drive/Outputs/Out/nCtrl5 <-> 3rd RxPDO Mapping/Mode Of Operation
//     Drive/Outputs/Out/nDataOut1 <-> 3rd RxPDO Mapping/Target Position
//     Drive/Outputs/Out/nDataOut2 <-> 3rd RxPDO Mapping/Target Velocity
//     Drive/Outputs/Out/nDataOut4[0] <-> 3rd RxPDO Mapping/Target Torque
//     Enc/Inputs/In/nDataIn1 <-> 3rd TxPDO Mapping/Actual Position
//     Enc/Inputs/In/nDataIn3 <-> 3rd TxPDO Mapping/Touch Probe Pos1 Pos Value
//     Enc/Inputs/In/nDataIn7 <-> 3rd TxPDO Mapping/Velocity actual value
//     Enc/Inputs/In/nDcInputTime <-> InfoData/DcInputShift
//     Enc/Inputs/In/nState4 @bit 1 <-> WcState/InputToggle
//     Enc/Inputs/In/nState4 <-> WcState/WcState
//     Enc/Inputs/In/nState5 <-> 3rd TxPDO Mapping/Touch Probe Status
//     Enc/Inputs/In/nState6 <-> 3rd TxPDO Mapping/Touch Probe Status @bit 8
//     Enc/Outputs/Out/nCtrl5 <-> 3rd RxPDO Mapping/Touch Probe Function
//     Enc/Outputs/Out/nCtrl6 <-> 3rd RxPDO Mapping/Touch Probe Function @bit 8
//   NC-Task 1 SAF/Axes/SpitUnit <-> Device 1 (EtherCAT)/Drive 27 (ASDA-A3-E CoE Drive)
//     Drive/Inputs/In/nDataIn3[0] <-> 2nd TxPDO Mapping/Actual Torque
//     Drive/Inputs/In/nDcOutputTime <-> InfoData/DcOutputShift
//     Drive/Inputs/In/nState1 <-> 2nd TxPDO Mapping/Status Word
//     Drive/Inputs/In/nState2 <-> 2nd TxPDO Mapping/Status Word @bit 8
//     Drive/Inputs/In/nState4 @bit 1 <-> WcState/InputToggle
//     Drive/Inputs/In/nState4 <-> WcState/WcState
//     Drive/Outputs/Out/nCtrl1 <-> 2nd RxPDO Mapping/Control Word
//     Drive/Outputs/Out/nCtrl2 <-> 2nd RxPDO Mapping/Control Word @bit 8
//     Drive/Outputs/Out/nDataOut1 <-> 2nd RxPDO Mapping/Target Position
//     Drive/Outputs/Out/nDataOut2 <-> 2nd RxPDO Mapping/Target Velocity
//     Drive/Outputs/Out/nDataOut4[0] <-> 2nd RxPDO Mapping/Target Torque
//     Enc/Inputs/In/nDataIn1 <-> 2nd TxPDO Mapping/Actual Position
//     Enc/Inputs/In/nDataIn3 <-> 2nd TxPDO Mapping/Touch Probe Pos1 Pos Value
//     Enc/Inputs/In/nDataIn7 <-> 2nd TxPDO Mapping/Velocity actual value
//     Enc/Inputs/In/nDcInputTime <-> InfoData/DcInputShift
//     Enc/Inputs/In/nState4 @bit 1 <-> WcState/InputToggle
//     Enc/Inputs/In/nState4 <-> WcState/WcState
//     Enc/Inputs/In/nState5 <-> 2nd TxPDO Mapping/Touch Probe Status
//     Enc/Inputs/In/nState6 <-> 2nd TxPDO Mapping/Touch Probe Status @bit 8
//     Enc/Outputs/Out/nCtrl5 <-> 2nd RxPDO Mapping/Touch Probe Function
//     Enc/Outputs/Out/nCtrl6 <-> 2nd RxPDO Mapping/Touch Probe Function @bit 8
//   NC-Task 1 SAF/Axes/Z_Axis <-> Device 1 (EtherCAT)/Drive 22 (ASDA-A3-E CoE Drive)
//     Drive/Inputs/In/nDataIn3[0] <-> 2nd TxPDO Mapping/Actual Torque
//     Drive/Inputs/In/nDcOutputTime <-> InfoData/DcOutputShift
//     Drive/Inputs/In/nState1 <-> 2nd TxPDO Mapping/Status Word
//     Drive/Inputs/In/nState2 <-> 2nd TxPDO Mapping/Status Word @bit 8
//     Drive/Inputs/In/nState4 @bit 1 <-> WcState/InputToggle
//     Drive/Inputs/In/nState4 <-> WcState/WcState
//     Drive/Outputs/Out/nCtrl1 <-> 2nd RxPDO Mapping/Control Word
//     Drive/Outputs/Out/nCtrl2 <-> 2nd RxPDO Mapping/Control Word @bit 8
//     Drive/Outputs/Out/nDataOut1 <-> 2nd RxPDO Mapping/Target Position
//     Drive/Outputs/Out/nDataOut2 <-> 2nd RxPDO Mapping/Target Velocity
//     Drive/Outputs/Out/nDataOut4[0] <-> 2nd RxPDO Mapping/Target Torque
//     Enc/Inputs/In/nDataIn1 <-> 2nd TxPDO Mapping/Actual Position
//     Enc/Inputs/In/nDataIn3 <-> 2nd TxPDO Mapping/Touch Probe Pos1 Pos Value
//     Enc/Inputs/In/nDataIn7 <-> 2nd TxPDO Mapping/Velocity actual value
//     Enc/Inputs/In/nDcInputTime <-> InfoData/DcInputShift
//     Enc/Inputs/In/nState4 @bit 1 <-> WcState/InputToggle
//     Enc/Inputs/In/nState4 <-> WcState/WcState
//     Enc/Inputs/In/nState5 <-> 2nd TxPDO Mapping/Touch Probe Status
//     Enc/Inputs/In/nState6 <-> 2nd TxPDO Mapping/Touch Probe Status @bit 8
//     Enc/Outputs/Out/nCtrl5 <-> 2nd RxPDO Mapping/Touch Probe Function
//     Enc/Outputs/Out/nCtrl6 <-> 2nd RxPDO Mapping/Touch Probe Function @bit 8
//   Clara_20230419/Clara_20230419 Instance <-> Device 1 (EtherCAT)/Drive 23 (ASDA-A3-E CoE Drive)
//     PlcTask Outputs/P_RollToRoll.Max_profile_velocity[1] <-> 3rd RxPDO Mapping/Max profile velocity
//   Clara_20230419/Clara_20230419 Instance <-> Device 1 (EtherCAT)/Drive 24 (ASDA-A3-E CoE Drive)
//     PlcTask Outputs/P_RollToRoll.Max_profile_velocity[3] <-> 3rd RxPDO Mapping/Max profile velocity
//   Clara_20230419/Clara_20230419 Instance <-> Device 1 (EtherCAT)/Drive 25 (ASDA-A3-E CoE Drive)
//     PlcTask Outputs/P_RollToRoll.Max_profile_velocity[2] <-> 3rd Receive PDO Mapping/Max profile velocity
//   Clara_20230419/Clara_20230419 Instance <-> Device 1 (EtherCAT)/Drive 26 (ASDA-A3-E CoE Drive)
//     PlcTask Outputs/P_RollToRoll.Max_profile_velocity[4] <-> 3rd RxPDO Mapping/Max profile velocity
//   Clara_20230419/Clara_20230419 Instance <-> Device 1 (EtherCAT)/Term 1 (EK1200)/Term 10 (EL1904)
//     PlcTask Inputs/.EL1904_M[2,{1..4}] <-> Module 1 (FSOES)/TxPDO/FSOE/InputChannel{1..4}  (4 links)
//   Clara_20230419/Clara_20230419 Instance <-> Device 1 (EtherCAT)/Term 1 (EK1200)/Term 11 (EL1904)
//     PlcTask Inputs/.EL1904_M[3,{1..4}] <-> Module 1 (FSOES)/TxPDO/FSOE/InputChannel{1..4}  (4 links)
//   Clara_20230419/Clara_20230419 Instance <-> Device 1 (EtherCAT)/Term 1 (EK1200)/Term 12 (EL1904)
//     PlcTask Inputs/.EL1904_M[4,{1..4}] <-> Module 1 (FSOES)/TxPDO/FSOE/InputChannel{1..4}  (4 links)
//   Clara_20230419/Clara_20230419 Instance <-> Device 1 (EtherCAT)/Term 1 (EK1200)/Term 13 (EL1904)
//     PlcTask Inputs/.EL1904_M[5,{1..4}] <-> Module 1 (FSOES)/TxPDO/FSOE/InputChannel{1..4}  (4 links)
//   Clara_20230419/Clara_20230419 Instance <-> Device 1 (EtherCAT)/Term 1 (EK1200)/Term 16 (EL2809)
//     PlcTask Outputs/.EL2809_M[4,{1..16}] <-> Channel {1..16}/Output  (16 links)
//   Clara_20230419/Clara_20230419 Instance <-> Device 1 (EtherCAT)/Term 1 (EK1200)/Term 17 (EL6001)
//     Task_com Inputs/.COMIN2/D[{0..21}] <-> COM Inputs/Data In {0..21}  (22 links)
//     Task_com Inputs/.COMIN2/Status <-> COM Inputs/Status
//     Task_com Outputs/.COMOUT2/Ctrl <-> COM Outputs/Ctrl
//     Task_com Outputs/.COMOUT2/D[{0..21}] <-> COM Outputs/Data Out {0..21}  (22 links)
//   Clara_20230419/Clara_20230419 Instance <-> Device 1 (EtherCAT)/Term 1 (EK1200)/Term 18 (EL6022)
//     PlcTask Inputs/P_Modbus_RTU.master[1].InData/D[{0..21}] <-> COM Inputs Channel 2/Data In {0..21}  (22 links)
//     PlcTask Inputs/P_Modbus_RTU.master[1].InData/Status <-> COM Inputs Channel 2/Status
//     PlcTask Outputs/P_Modbus_RTU.master[1].OutData/Ctrl <-> COM Outputs Channel 2/Ctrl
//     PlcTask Outputs/P_Modbus_RTU.master[1].OutData/D[{0..21}] <-> COM Outputs Channel 2/Data Out {0..21}  (22 links)
//     Task_com Inputs/.COMIN1/D[{0..21}] <-> COM Inputs Channel 1/Data In {0..21}  (22 links)
//     Task_com Inputs/.COMIN1/Status <-> COM Inputs Channel 1/Status
//     Task_com Outputs/.COMOUT1/Ctrl <-> COM Outputs Channel 1/Ctrl
//     Task_com Outputs/.COMOUT1/D[{0..21}] <-> COM Outputs Channel 1/Data Out {0..21}  (22 links)
//   Clara_20230419/Clara_20230419 Instance <-> Device 1 (EtherCAT)/Term 1 (EK1200)/Term 2 (EL1809)
//     PlcTask Inputs/.EL1809_M[1,{1..16}] <-> Channel {1..16}/Input  (16 links)
//   Clara_20230419/Clara_20230419 Instance <-> Device 1 (EtherCAT)/Term 1 (EK1200)/Term 3 (EL1809)
//     PlcTask Inputs/.EL1809_M[2,{1..16}] <-> Channel {1..16}/Input  (16 links)
//   Clara_20230419/Clara_20230419 Instance <-> Device 1 (EtherCAT)/Term 1 (EK1200)/Term 4 (EL1809)
//     PlcTask Inputs/.EL1809_M[3,{1..16}] <-> Channel {1..16}/Input  (16 links)
//   Clara_20230419/Clara_20230419 Instance <-> Device 1 (EtherCAT)/Term 1 (EK1200)/Term 5 (EL2809)
//     PlcTask Outputs/.EL2809_M[1,{1..16}] <-> Channel {1..16}/Output  (16 links)
//   Clara_20230419/Clara_20230419 Instance <-> Device 1 (EtherCAT)/Term 1 (EK1200)/Term 6 (EL2809)
//     PlcTask Outputs/.EL2809_M[2,{1..16}] <-> Channel {1..16}/Output  (16 links)
//   Clara_20230419/Clara_20230419 Instance <-> Device 1 (EtherCAT)/Term 1 (EK1200)/Term 7 (EL2809)
//     PlcTask Outputs/.EL2809_M[3,{1..16}] <-> Channel {1..16}/Output  (16 links)
//   Clara_20230419/Clara_20230419 Instance <-> Device 1 (EtherCAT)/Term 1 (EK1200)/Term 8 (EL6900)
//     PlcTask Inputs/P_TwinSAFE.Com_err <-> StandardInputs/Standard Out Var 46
//     PlcTask Inputs/P_TwinSAFE.FB_err <-> StandardInputs/Standard Out Var 47
//     PlcTask Inputs/P_TwinSAFE.TwinSAFE_Group_State <-> TwinSAFE Group Info Data/TwinSafeGroup1 Info Data/State
//     PlcTask Outputs/P_TwinSAFE.Err_Ack <-> StandardOutputs/Standard In Var 39
//   Clara_20230419/Clara_20230419 Instance <-> Device 1 (EtherCAT)/Term 1 (EK1200)/Term 9 (EL1904)
//     PlcTask Inputs/.EL1904_M[1,{1..4}] <-> Module 1 (FSOES)/TxPDO/FSOE/InputChannel{1..4}  (4 links)
//   Clara_20230419/Clara_20230419 Instance <-> Device 1 (EtherCAT)/Term 28 (EK1100)/Term 29 (EL1809)
//     PlcTask Inputs/.EL1809_S[1,{1..16}] <-> Channel {1..16}/Input  (16 links)
//   Clara_20230419/Clara_20230419 Instance <-> Device 1 (EtherCAT)/Term 28 (EK1100)/Term 30 (EL1809)
//     PlcTask Inputs/.EL1809_S[2,{1..16}] <-> Channel {1..16}/Input  (16 links)
//   Clara_20230419/Clara_20230419 Instance <-> Device 1 (EtherCAT)/Term 28 (EK1100)/Term 31 (EL2809)
//     PlcTask Outputs/.EL2809_S[1,{1..16}] <-> Channel {1..16}/Output  (16 links)
//   Clara_20230419/Clara_20230419 Instance <-> Device 1 (EtherCAT)/Term 28 (EK1100)/Term 32 (EL4002)
//     PlcTask Outputs/.EL4002_S[1] <-> AO Outputs Channel 1/Analog output
//     PlcTask Outputs/.EL4002_S[2] <-> AO Outputs Channel 2/Analog output
//   Clara_20230419/Clara_20230419 Instance <-> NC-Task 1 SAF/Axes/Axis_FS
//     PlcTask Inputs/.Axis[1].Ref.NcToPlc <-> Outputs/ToPlc
//     PlcTask Outputs/.Axis[1].Ref.PlcToNc <-> Inputs/FromPlc
//   Clara_20230419/Clara_20230419 Instance <-> NC-Task 1 SAF/Axes/Axis_SS
//     PlcTask Inputs/.Axis[2].Ref.NcToPlc <-> Outputs/ToPlc
//     PlcTask Outputs/.Axis[2].Ref.PlcToNc <-> Inputs/FromPlc
//   Clara_20230419/Clara_20230419 Instance <-> NC-Task 1 SAF/Axes/Axis_unwider_input1
//     PlcTask Inputs/P_RollToRoll.FB_RoolToRool[1].REF.NcToPlc <-> Outputs/ToPlc
//     PlcTask Outputs/P_RollToRoll.FB_RoolToRool[1].REF.PlcToNc <-> Inputs/FromPlc
//   Clara_20230419/Clara_20230419 Instance <-> NC-Task 1 SAF/Axes/Axis_unwinder_input2
//     PlcTask Inputs/P_RollToRoll.FB_RoolToRool[3].REF.NcToPlc <-> Outputs/ToPlc
//     PlcTask Outputs/P_RollToRoll.FB_RoolToRool[3].REF.PlcToNc <-> Inputs/FromPlc
//   Clara_20230419/Clara_20230419 Instance <-> NC-Task 1 SAF/Axes/Axis_winder_output1
//     PlcTask Inputs/P_RollToRoll.FB_RoolToRool[2].REF.NcToPlc <-> Outputs/ToPlc
//     PlcTask Outputs/P_RollToRoll.FB_RoolToRool[2].REF.PlcToNc <-> Inputs/FromPlc
//   Clara_20230419/Clara_20230419 Instance <-> NC-Task 1 SAF/Axes/Axis_winder_output2
//     PlcTask Inputs/P_RollToRoll.FB_RoolToRool[4].REF.NcToPlc <-> Outputs/ToPlc
//     PlcTask Outputs/P_RollToRoll.FB_RoolToRool[4].REF.PlcToNc <-> Inputs/FromPlc
//   Clara_20230419/Clara_20230419 Instance <-> NC-Task 1 SAF/Axes/SpitUnit
//     PlcTask Inputs/.Axis[4].Ref.NcToPlc <-> Outputs/ToPlc
//     PlcTask Outputs/.Axis[4].Ref.PlcToNc <-> Inputs/FromPlc
//   Clara_20230419/Clara_20230419 Instance <-> NC-Task 1 SAF/Axes/Z_Axis
//     PlcTask Inputs/.Axis[3].Ref.NcToPlc <-> Outputs/ToPlc
//     PlcTask Outputs/.Axis[3].Ref.PlcToNc <-> Inputs/FromPlc

CONFIGURATION Clara_20230419
    RESOURCE PLC ON TwinCAT3
        TASK PlcTask(INTERVAL := T#10ms, PRIORITY := 12);
        TASK Task_com(INTERVAL := T#2ms, PRIORITY := 6);
        PROGRAM MAIN WITH PlcTask : MAIN;
        PROGRAM PRG_COMM WITH Task_com : PRG_COMM;
    END_RESOURCE
END_CONFIGURATION

// ---- DUTs/01_ST_IO/ST_Input.TcDUT
TYPE ST_Input :
STRUCT
(****************XYZ,用io.********************)	
	
(****************ISS********************)
	biSubInkTankLevel				:ARRAY[1..20] OF BOOL;	//
	(*
			墨桶	液位	泵		
1	LC	1,2	1,2	FB_SubInkFeed_C	[1]
2	LM	3,4	3,4	FB_SubInkFeed_C	[2]
3	Y	5,6	5,6	FB_SubInkFeed_C	[3]
4	M	7,8	7,8	FB_SubInkFeed_C	[4]
5	C	9,10	9,10	FB_SubInkFeed_C	[5]
6	K	11,12	11,12	FB_SubInkFeed_C	[6]
7	W	13,14,15,16	13,15	FB_SubInkFeed_W	
8	P	17,18	17,18	FB_SubInkFeed_P	
9	F	19,20	19,20	FB_SubInkFeed_Flush	

	*)
	
	biProtectAirTankLevel_C			:BOOL;	//保护气瓶液位
	biProtectAirTankLevel_W			:BOOL;	//保护气瓶液位
	btPurge									:BOOL;//正压按钮
	btVacBt_W								:BOOL;//白墨，负压按钮
	btVacBt_C								:BOOL;//彩墨，负压按钮
(****************测高********************)
	biElectromagnet_limit			:BOOL;	
(****************UpDownSlot********************)
	biUDS_sensor_up_S					:ARRAY[1..number_UpDownSlot] OF BOOL;  //s1-s6
	biUDS_sensor_down_S1				:ARRAY[1..16] OF BOOL;//s1
(****************FootPedal********************)	
	biFootPedal						:ARRAY[1..number_FootPedal] OF ST_IO_FootPedal;
(****************RoolToRool********************)	
	biDualSensor					:ARRAY[1..2] OF BOOL;
	biClamp_hold					:ARRAY[1..2] OF BOOL;//卡箍抱紧
	biBrakeBack_L					:BOOL;//左刹车反馈
	biBrakeBack_R					:BOOL;//右刹车反馈
	
(****************safe********************)	
	biRely_back  											:ARRAY[1..4] OF BOOL;
	btReset													:BOOL;

	
END_STRUCT
END_TYPE

// ---- DUTs/01_ST_IO/ST_IO_FootPedal.TcDUT
TYPE ST_IO_FootPedal :
STRUCT
	PedalPressed1			:BOOL;	//LEFT
	PedalPressed2			:BOOL;	//MID
	PedalPressed3			:BOOL;	//RIGHT
END_STRUCT
END_TYPE

// ---- DUTs/02_PLC/stAxis.TcDUT
TYPE stAxis :
STRUCT	
(*******************C#API*************************************************)
//R//
	Error								:BOOL;
	ErrorId							  	:UDINT;	//
	Home_Done					:BOOL;
	Move_Done					:BOOL;
	state							  	 :INT; //
	position							 :LREAL;//um		The actual position of the drive
	LimitN                             :BOOL; //负极限
	LimitP                             :BOOL; //正极限
    Origin                            :BOOL; //原点
	AxisErrorId					 :UDINT;// 轴错误
	ControlLoopClosed				 :BOOL;//使能
//W//	
	Enabled		                      :BOOL; 	//伺服ON	
	Disable							  :BOOL;//伺服Off
	velocity							  :LREAL;//mm/s
	acceleration					  :LREAL:=5709;//	mm/s2		
	jerk								  :LREAL:=28591;//mm/s3
	homeoffset					  :LREAL:=10;//mm
	homingvelocity				  :LREAL:=5;//mm/s   The velocity used during homing
	requestedposition			  :LREAL;//um		The position to move to absolutely
	requestedoffset				  :LREAL;//um		The distance to move over relatively	
	constantvelocitystart		  :LREAL;//um		The position to start moving with a constant velocity
												//      0 < ConstantVelocityStart< ConstanVelocityEnd< RequestedPosition
	constanvelocityend			  :LREAL;//um		The position to end moving with a constant velocity	
	homingtimeout				  :LREAL:=60;//s    A timeout that overrules the default
	maxDistance					  :LREAL:=3000;	//mm 	The maximal mechanical distance that can be moved safely
	stop								  :BOOL;//
	reset								  :BOOL;//
	Initialize							  :BOOL;//
	MoveConstantVelocity	  :BOOL;//
	HomeExe						  :BOOL;//
	MoveAbsoluteExe			  :BOOL;//
	MoveRelativeExe			  :BOOL;//
	MoveVelocityExe			  :BOOL;//
	JogForward					  :BOOL;//
	JogBackwards				  :BOOL;//
	Setoff							  :BOOL;
	Automatic_positioning	  :BOOL;//自动测高
	commandtimeout			 :LREAL:=10;//s		
END_STRUCT
END_TYPE

// ---- DUTs/02_PLC/stISS.TcDUT
TYPE stISS :
STRUCT
	//R//						
		error_code			:INT;
		state						:INT;
		mainTankLevel		:LREAL;
		Init_Done				:BOOL;
		Error						:BOOL;
	//W//
		Initialize				:BOOL;	//  
		Setoff				:BOOL;	//  
		sensor_blink		:BOOL;
END_STRUCT
END_TYPE

// ---- DUTs/02_PLC/stSubTank.TcDUT
TYPE stSubTank :
STRUCT
	//R//						
		error_code			:INT;
		state				:INT;
		Error				:BOOL;
	//W//
		Setoff				:BOOL;	//  
END_STRUCT
END_TYPE

// ---- DUTs/02_PLC/stRtu.TcDUT
TYPE stRtu :
STRUCT
	_01b_writearray:ARRAY [1..10] OF BYTE;//modsim 01口写操作数组（bool）
	_01b_readarray:ARRAY [1..10] OF BYTE;//modsim 01口读操作数组（bool）
    _02OR_array :ARRAY [1..10] OF BYTE;//modsim 02口读操作数组
	_03writearray:ARRAY [1..10] OF WORD;//modsim 03口写操作数组
	_03readarray:ARRAY [1..10] OF WORD;//modsim 03口读操作数组
	_04readarray:ARRAY[1..10] OF WORD;//04口 读	
	_06writesinglearray:ARRAY [1..10] OF WORD;//modsim 06口写操作数组
	_06writesinglearray_PID:ARRAY [1..6] OF WORD:=[10,10];//modsim 06口写操作数组
END_STRUCT
END_TYPE

// ---- DUTs/02_PLC/stSpitUnit.TcDUT
TYPE stSpitUnit  :
STRUCT
//R//
	error_code					:UDINT;
	state						:INT;
	home_sensor_covered			:BOOL;
	current_position			:LREAL;
	AxisErrorId					:UDINT;
	Home_Done					:BOOL;
	Move_Done					:BOOL;
	Error								:BOOL;
	Homing							:BOOL;
	ControlLoopClosed				 :BOOL;//使能
//W//	
	acceleration				:LREAL;
	moving_speed_up				:LREAL:=5;
	moving_speed_down				:LREAL:=5;	
	target_position				:LREAL;	
	spindle_length				:LREAL:=50;
	FanState					:BOOL;
	Initialize					:BOOL;
	HomeExe						:BOOL;
	MoveAbsoluteExe				:BOOL;
	SetOff						:BOOL;

END_STRUCT
END_TYPE

// ---- DUTs/02_PLC/stTableVacuum.TcDUT
TYPE stTableVacuum :
STRUCT
//R//
	error_code					:INT;	//	
	state					:INT;	//	
	vacuum_measured			:LREAL;//	Pa
	Error                :BOOL;
//W//	
	vacuum_min				:LREAL:=0;	//	Pa 3.5
	vacuum_max				:LREAL:=10;	//	Pa	10
	setpoint				:LREAL:=6;	//	Pa	6[0-8]
	vacuum_offset_collector	:LREAL;	//	Pa	Offset used to calibrate the vacuum sensor of the vacuum collector
	setpoint_range_pct		:LREAL:=70;	//	%  Threshold used to indicate the table vacuum is ready
	vacuum_timeout			:LREAL:=60000;	//ms	TIME needed TO reach the vacuum setpoint.
	vacuum_off_timeout		:LREAL:=30000;	//	ms 	Time to turn off the vacuum
	
	Initialize				:BOOL;
	SetVacuumOn				:BOOL;
	SetVacuumOff			:BOOL;
	Setoff					:BOOL;
	ctrlP						: LREAL:=10;//制冷比例
	ctrlI						: LREAL;//制冷积分
	ctrlD						: LREAL;//制冷微分
	
END_STRUCT
END_TYPE

// ---- DUTs/02_PLC/stUVLed.TcDUT
TYPE stUVLed :
STRUCT
//R//
	error_code					:INT;
	state					:INT;
	initialized			:BOOL;
	settings_applied		:BOOL;
	curing_started	:BOOL;
	curing_stopped	:BOOL;
	error					:BOOL;
	off					:BOOL;
//W//	
	unidirection			:BOOL;//"(ConfigurePowerSettings parameter)Indicates unidirectional printing.TRUE IF the print is unidirectional, otherwise FALSE FOR bi-directional printing.
	initial_print_position	:INT;//"(ConfigurePowerSettings parameter)Indicates the initial print position: 0:from_home, 1:to_home."
	uv_power_leading		:DINT;//% "(leadingPower ConfigurePower-Settings method)Power to apply to leading LEDs of the UVUnit"
	uv_power_trailing		:DINT;//% "(trailingPower ConfigurePower-Settings method)Power to apply to trailing LEDs of the UVUnit"
	uvStart					:LREAL;//mm "Position in micron where to start/stop curing depending on the direction (left/right)."
	uvEnd					:LREAL;//mm "Position in micron where to start/stop curing depending on the direction (left/right)"
	
	Initialize				:BOOL;
	ConfigurePowerSettings	:BOOL;
	ConfigurePositions		:BOOL;
	StopCuring				:BOOL;
	SetOff					:BOOL;
	prats				    :BYTE:=16#3F;//分段开灯，1-6,6为全开
	ahead_pos				:LREAL:=100;//因YV灯有延迟，提前量
	delay_pos				:LREAL:=100;//因YV灯有延迟，关闭延时
END_STRUCT
END_TYPE

// ---- Enum_Text/Enum/PLC/AxisStateEnum.TcDUT
{attribute 'qualified_only'}
{attribute 'strict'}
{attribute 'to_string'}
TYPE AxisStateEnum :
(
	off			:=	0	,//	The Reset command finished successful
	idle		:=	1	,//	The Initialize command finished successful
	homing		:=	2	,//	The Home command started successful. The drive is moving
	ready		:=	3	,//	The Home command finished successful and the drive is idle again. Or The MoveX commands finished successful and the drive is idle again
	moving		:=	4	,//	The MoveX command started successful. The drive is moving
	stopping	:=	5	,//	The axis object is stopping
	disabled	:=	6	,//	The axis object  is disabled
	error		:=	100	//	The axis object  is in error state

);
END_TYPE

// ---- Enum_Text/Enum/PLC/Axis_XY_ErrorEnum.TcDUT
{attribute 'qualified_only'}
{attribute 'strict'}
{attribute 'to_string'}
TYPE Axis_XY_ErrorEnum :
(
no_error	:=	0	,//	No error detected
not_connected	:=	1	,//	A command was requested prior to opening the driver
invalid_state	:=	2	,//	An invalid command was requested
actuator_out_of_pos_range	:=	3	,//	?
actuator_out_of_neg_range	:=	4	,//	?
homing_timeout	:=	5	,//	
parameter_out_of_range	:=	6	,//	
trigger_Limit	:=	7	,//	limit is triggered
SpeedNotReach	:=	8	,//	command "MoveConstantVelocity" is not reach set speed 
homing_error	:=	9	,//	The homing sequence failed 
cmd_timeout	:=	10	,//	Emstop is trigger
TBD_error	:=	11	,//	
io_error	:=	12	,//	IO error HW board
unknown_error	:=	13	,//	Unknown – Network error
Drive_not_ready_for_operation	:=	14	,//	Drive not ready for operation
interlock_error	:=	15	,//
Invalid_IO_data_for_more_than_n_subsequent_NC_cycles_encoder	:=	16	,//	Possible reasons for this error: An EtherCAT slave may have left its OP state or there is a too high real time usage or a too high real time jitter.

emergency_error	:=	666	//	


	
);
END_TYPE

// ---- Enum_Text/Enum/PLC/FootPedalErrorEnum.TcDUT
{attribute 'qualified_only'}
{attribute 'strict'}
{attribute 'to_string'}
TYPE FootPedalErrorEnum :
(
no_error	:=	0	,//	No error detected
not_connected	:=	1	,//	A command was requested prior to opening the driver
invalid_state	:=	2	,//	An invalid command was requested
io_error	:=	3	,//	IO error HW board
unknown_error	:=	4	,//	Unknown / Network error
emergency_error	:=	666	//	


);
END_TYPE

// ---- Enum_Text/Enum/PLC/FootPedalStateEnum.TcDUT
{attribute 'qualified_only'}
{attribute 'strict'}
{attribute 'to_string'}
TYPE FootPedalStateEnum :
(
	ready	:=	0	,//	The FootPedal is in ready-state.
	error	:=	100	//	The FootPedal is in error.

);
END_TYPE

// ---- Enum_Text/Enum/PLC/ISSErrorEnum.TcDUT
{attribute 'qualified_only'}
{attribute 'strict'}
{attribute 'to_string'}
TYPE ISSErrorEnum :
(
no_error	:=	0	,//	No error detected
not_connected	:=	1	,//	A command was requested prior to opening the driver
invalid_state	:=	2	,//	An invalid command was requested
pump1_failure	:=	4	,//	Pump1 is in error
pump2_failure	:=	6	,//	Pump2 is in error
back_to_air_tank	:=	8	,//	
io_error	:=	9	,//	
unknown_error	:=	10	,//	
emergency_error	:=	666	//	



);
END_TYPE

// ---- Enum_Text/Enum/PLC/SubTankInkEnum.TcDUT
{attribute 'qualified_only'}
{attribute 'strict'}
{attribute 'to_string'}
TYPE SubTankInkEnum :
(
circuit_not_filled			:=	0	,//	0” circuit not filled (default setting)
white_ink					:=	1	,//	“1” circuit filled with “white ink”
storage_flush				:=	2	//	“2” circuit filled with “storage fluid”

);
END_TYPE

// ---- Enum_Text/Enum/PLC/SubTankStateEnum.TcDUT
{attribute 'qualified_only'}
{attribute 'strict'}
{attribute 'to_string'}
TYPE SubTankStateEnum :
(

ready	:=	0	,//	
error	:=	100	//	


);
END_TYPE

// ---- Enum_Text/Enum/PLC/MUErrorEnum.TcDUT
{attribute 'qualified_only'}
{attribute 'strict'}
{attribute 'to_string'}
TYPE MUErrorEnum :
(
no_error									:=	0	,//	No error detected
not_connected							:=	1	,//	A command was requested prior to opening the driver
invalid_state								:=	2	,//	An invalid command was requested
alarm_circulation_left					:=	3	,//	When pump 3 was activate less than …x/min => 
alarm_circulation_right				:=	4	,//	When pump 6 was activate less than …x/min => 
alarm_through_left						:=	5	,//	When pump 3 was activate less than 1x/2min =>
alarm_through_right					:=	6	,//	When pump 6 was activate less than 1x/2min => 
alarm_runtime_circulation_left		:=	7	,//	When pump 3 runs longer than 8sec => 
alarm_runtime_circulation_right	:=	8	,//	When pump 6 runs longer than 8sec => 
unknown_error							:=	9	,//	Unknown – Network error
emergency_error						:=	666	//	The object is in error due to an active emergency error.


	
);
END_TYPE

// ---- Enum_Text/Enum/PLC/MUStateEnum.TcDUT
{attribute 'qualified_only'}
{attribute 'strict'}
{attribute 'to_string'}
TYPE MUStateEnum :
(
off	:=	0	,//	The MaintenanceUnit is in off-state.
idle	:=	1	,//	The MaintenanceUnit is in idle-state.
swapping	:=	2	,//	The MaintenanceUnit is busy swapping fluids
error	:=	100	//	The MaintenanceUnit is in error.


);
END_TYPE

// ---- Enum_Text/Enum/PLC/SwapInfoEnum.TcDUT
{attribute 'qualified_only'}
{attribute 'strict'}
{attribute 'to_string'}
TYPE SwapInfoEnum :
(
NONE	:=	0	,//	
AC_STORAGE_FLUSH_RUNS	:=	1	,//
AC_STORAGE_FLUSH_NEEDS_HELP	:=	2	,//
AC_STORAGE_FLUSH_FINISHED	:=	3	,//
AC_WHITE_INK_RUNS	:=	4	,//
AC_WHITE_INK1_NEEDS_HELP	:=	5	,//
AC_WHITE_INK2_NEEDS_HELP	:=	6	,//
AC_WHITE_INK_FINISHED	:=	7	//



	
);
END_TYPE

// ---- Enum_Text/Enum/PLC/TabVacStateEnum.TcDUT
{attribute 'qualified_only'}
{attribute 'strict'}
{attribute 'to_string'}
TYPE TabVacStateEnum :
(
	off					:=	0	,//	The TableVacuum is in off-state.
	idle				:=	1	,//	The TableVacuum is in idle-state.
	waiting_vacuum_on	:=	2	,//	The TableVacuum object is waiting until the vacuum pressure is reached.
	waiting_vacuum_off	:=	3	,//	The TableVacuum object is waiting until the vacuum pressure is dropped.
	on					:=	4	,//	The TableVacuum is on.
	waiting_off			:=	5	,//	The TableVacuum  is waiting to switched off.
	error				:=	100	//	The TableVacuum is in error.

);
END_TYPE

// ---- Enum_Text/Enum/TwinSafe/TwinSAFE_FB_ESTOP_State_Enum.TcDUT
{attribute 'qualified_only'}
{attribute 'strict'}
{attribute 'to_string'}
TYPE TwinSAFE_FB_ESTOP_State_Enum :
(
	undefined	:=	0	,(*	undefined	*)
RUN	:=	1	,(*	"RUN
The FB ESTOP module assumes the RUN state if no error is present and no active EStopIn
input requests a safe state.
The outputs assume the following values:
Error=0
EStopOut=1
EStopDelOut=1"	*)
STOP	:=	2	,(*	"STOP
The FB ESTOP module assumes the STOP state if the input FbRun is FALSE.
The outputs assume the following values:
Error=0
EStopOut=0
EStopDelOut=0"	*)
SAFE	:=	3	,(*	"SAFE
The FB ESTOP module assumes the SAFE state as long as at least one of the active
EStopIn inputs has requested the safe state.
The outputs assume the following values:
Error=0
EStopOut=0
EStopDelOut=0"	*)
ERROR	:=	4	,(*	"ERROR
If the FB ESTOP module detects an error, the FB ESTOP module assumes the ERROR state
and transmits the corresponding Diag message to the GROUP module.
The outputs assume the following values:
Error=1
EStopOut=0
EStopDelOut=0"	*)
RESET	:=	5	,(*	"RESET
The FB ESTOP module assumes the RESET state if no further error is pending after an
error has occurred and the ErrAck input of the corresponding group is set to TRUE.
The outputs assume the following values:
Error=0
EStopOut=0
EStopDelOut=0"	*)
START	:=	6	,(*	"START
The FB ESTOP module assumes the START state if the Restart input is TRUE, in order to
wait for a rising and falling edge of the Restart input before entering the RUN state and the
outputs leave the safe state.
The outputs assume the following values:
Error=0
EStopOut=0
EStopDelOut=0"	*)
DELAYOUT	:=	8	(*	"DELAYOUT
The FB ESTOP module assumes the DELAYOUT state if at least one of the active EStopIn
inputs has requested the safe state and the delay time for the EStopDelOut output has not
yet expired.
The outputs assume the following values:
Error=0
EStopOut=0
EStopDelOut=1"	*)

);
END_TYPE

// ---- POUs/000_程序辅助系统/报警/Data types/Alm_AlarmType.TcDUT
TYPE Alm_AlarmType :
STRUCT
      (*InPut*)
	EventId:					DINT;
    EventMessage:			WSTRING(255);//报警时间+等级+内容
    EventTime:                   DT;
	EventActive:				BOOL;
	QuitRequired:				BOOL;
	QuitEvent:				BOOL;
	EventClass:				Alm_EventClass;
	AlarmMsg:				Alm_AlmMsg;
	AlarmlampOn:			BOOL;(*报警灯*)
	AutoRunOff:				BOOL;(*退出自动循环*)

	(* event actions OutPut	*)
	AlarmAction1:				BOOL;
	AlarmAction2:				BOOL;
	AlarmAction3:				BOOL;
	AlarmAction4:				BOOL;
	AlarmAction5:				BOOL;
	AlarmAction6:				BOOL;
	AlarmAction7:				BOOL;
	AlarmAction8:				BOOL;

       (*OutPut*)
	EventAlive:					BOOL;
    ShowlampOn:           		BOOL;
	InUse:                		BOOL;
END_STRUCT
END_TYPE;

// ---- POUs/000_程序辅助系统/报警/Data types/Alm_AlmMsg.TcDUT
TYPE Alm_AlmMsg :
STRUCT
	CN:		WSTRING(255):="中文";
	EN:		STRING(255):='En';	
END_STRUCT
END_TYPE

// ---- POUs/000_程序辅助系统/报警/Data types/Alm_EventClass.TcDUT
{attribute 'qualified_only'}
{attribute 'strict'}
{attribute 'to_string'}
TYPE Alm_EventClass :
(
    NoAlarm        :=0,(*无警报*)
    Message      :=1,(*信息*)
    Event        :=2,(*事件*)
    non_3          :=3,(*暂无*)
    non_4          :=4,(*暂无*)
    non_5          :=5,(*暂无*)
    Alarm        :=6,(*不停机警报*)
    Stop         :=7(*停机警报*)
);
END_TYPE

// ---- Global Variables/_01_Global_Variables.TcGVL
{attribute 'Tc2GvlVarNames'}
VAR_GLOBAL
	Axis:                   ARRAY[1..4] OF 	Axis_PTP_CoE;(*1:FastScan; 2:SlowScan; 3:Z_Axis; 4:SpitUnit*)
			
END_VAR

VAR_GLOBAL PERSISTENT(*断电保存型变量*)
	
	State_reset_time			:TIME:=T#100MS;//状态自复位延时时间
	inkFillTimeOutSet  		:TIME:=T#60S;
	T								:ARRAY[1..13] OF LREAL:=[45,4,0.5,15,120,0.2,1,60,180,2,240,1200,100];
	
	(******************drip_purge,接收上位数据，并保存***********************)
	IntervalTime_W 			:LREAL;//min
	DripTime_W 				:LREAL;//sec
	PurgeTime_W 			:LREAL;//sec
	IntervalTime_C 			:LREAL;//min
	DripTime_C 				:LREAL;//sec
	PurgeTime_C 			:LREAL;//sec
	(**********************墨盒里 
		0” circuit not filled (default setting)
	“1” circuit filled with “white ink”
	“2” circuit filled with “storage fluid”
	****)
	SubTankInk_type			:INT;//


(***********************HMI******************************)	
	HMI_SetStirrer_continueTime			:LREAL:=0.1;//M   持续时间
	HMI_SetStirrer_intervalTime			:LREAL:=5;//M  间隔时间
	HMI_SetWaste_continueTime			:LREAL:=0.1;//M   废墨持续时间
	HMI_SetWaste_intervalTime			:LREAL:=5;//M  废墨间隔时间
	HMI_CircPump1_V						:LREAL:=1;(*0-5V*)
	HMI_CircPump2_V						:LREAL:=1;(*0-5V*)
	HMI_EM_STOP_Dec_FS					:LREAL:=5709;
	HMI_EM_STOP_Jerk_FS					:LREAL:=28591;
	
	HMI_RTR_set_Torque          		:ARRAY[1..4] OF DINT:=[80,80,80,80];//0-100
	
	HMI_Vac_dely_on						:INT:=3000;//ms
	
	
	
	
END_VAR

VAR_GLOBAL CONSTANT
	FastScan:INT:=1;
	SlowScan:INT:=2;
	Z_Axis	:INT:=3;
	SpitUnit :INT:=4;
	number_TableVacuum:INT:=1;
	number_UpDownSlot:INT:=6;	//1-6  S1-S6
	number_FootPedal:INT:=4;	//1-4:1-4:1:Footpedal1 input; 2:Footpedal2 output; 3:Footpeda3  input; 4:Footpedal4 output
	number_RoolToRool:INT:=4;   //1:input1; 2:output1; 3:input2; 4:output2
END_VAR

// ---- Global Variables/_04_Global_Variables_InOutput.TcGVL
{attribute 'Tc2GvlVarNames'}
VAR_GLOBAL(*输入输出*)

	(*程序用变量*)
	stInput					:ST_Input;
	stOutput				:ST_Output;

	
	(*链接到硬件的变量*)
	EL1809_M AT%I*			:ARRAY[1..3,1..16] OF BOOL;
	EL2809_M AT%Q*			:ARRAY[1..4,1..16] OF BOOL;
	EL1904_M AT%I*			:ARRAY[1..5,1..4] OF BOOL;
	
	
	EL1809_S AT%I*			:ARRAY[1..2,1..16] OF BOOL;
	EL2809_S AT%Q*			:ARRAY[1..1,1..16] OF BOOL;
	EL4002_S AT%Q*			:ARRAY[1..2] OF INT;
	
	(*******************SafetyGuard*****************)
	EL2904 					:ARRAY[1..3,1..4] OF BOOL;
	
END_VAR

// ---- GVLs/COMM.TcGVL
{attribute 'Tc2GvlVarNames'}
VAR_GLOBAL
	COMCONTROL1,COMCONTROL2   :SerialLineControl;  //串行通讯的功能块 
    COMIN1,COMIN2 	 AT%I*	  :KL6inData22B;      //22字节的IO端子模式
    COMOUT1,COMOUT2  AT%Q*	  :KL6outData22B;     
    TXBUFFER1		  :COMBUFFER;
    TXBUFFER2		  :COMBUFFER;    //串口通讯的缓存
    RXBUFFER1		  :COMBUFFER;
    RXBUFFER2		  :COMBUFFER;//说明：不论什么类型的硬件接口,Buffer变量类型都为ComBufferfer
                                     //其中包括了 300字节的缓存区和一些状态参数标志位。
END_VAR

// ---- GVLs/GVL.TcGVL
{attribute 'qualified_only'}
VAR_GLOBAL
(********************ISS****************************)	
		MainTankLevel		:ARRAY[1..10] OF LREAL; //LC,LM,Y,M,C,K,W,P,F,WAST
		MainTankLevel_timeout:BOOL;
		inkLevel_W_L_BOT	:BOOL;
		inkLevel_W_L_TOP	:BOOL;
		inkLevel_W_R_TOP	:BOOL;
		inkLevel_W_R_BOT	:BOOL;	
		fill_W_in_swap_enable	:BOOL;
		fill_F_in_swap_enable	:BOOL;
(**************UVLED********************)
	set_uv_power_left		:DINT;//set power
	set_uv_power_right		:DINT;//set power
	set_uv_parts_left		:BYTE;
	set_uv_parts_right		:BYTE;
	HMI_TEMP_L,HMI_TEMP_R :INT;
	HMI_power_L,HMI_power_R:INT;
	UV_error_L,UV_error_R:BOOL;
	UV_timeout:BOOL;
	UVisRemote:BOOL;//远程模式	
(******************System*************************)
	temp_measured:LREAL;
	humidity_measured:LREAL;
(********************safe****************************)	
		Emstop_SAFE			:BOOL;		//急停 安全输出
		Emstop_Button		:BOOL;		//急停按 钮
		Reset			:BOOL;
		shuttle_crash		:BOOL;		//碰撞
		interlock_triggered		:BOOL;	//	安全门触发
		
(*********************)
	HMI_btReset				:BOOL;
	HMI_btEmstop		:BOOL;	
END_VAR

// ---- GVLs/GVL_Alarm.TcGVL
VAR_GLOBAL
		gbAlarm_NoStopAlarm,
		gbAlarm_StopAlarm ,
		gbAlarm_ShowlampOn ,
		gbAlarm_FalshLamp ,
		gbAlarm_NeedPause ,
		gbAlarm_ExtruderOff ,
		gbAlarm_HydraulicOff ,
		gbAlarm_HeatingOff ,
		gbAlarm_FillingOff ,
		gbAlarm_ServoMotorOff ,
		gbAlarm_AutoRunOff ,
		gbAlarm_AlarmAction1 ,
		gbAlarm_AlarmAction2 ,
		gbAlarm_AlarmAction3 ,
		gbAlarm_AlarmAction4 ,
		gbAlarm_AlarmAction5 ,
		gbAlarm_AlarmAction6 ,
		gbAlarm_AlarmAction7 ,
		gbAlarm_AlarmAction8	:			BOOL;
		
	  	Alm_ActiveAlarmNum:      DINT;(*当前激活警报的数量*)
	 	Alm_HistoryAlarmNum:     DINT;(*历史警报的数量*)
	 	AlarmActionArray:		 ARRAY [cnAlarmFirst..cnAlarmLast] OF Alm_AlarmType;(*记录所有警报状态的数组*)
		AlarmActiveArray:		 ARRAY [cnAlmActiveFirst..cnAlmActiveLast] OF Alm_AlarmHistoryType;(*记录已激活警报状态的数组*)
		fbSetAlarm:				 ARRAY[cnAlarmFirst..cnAlarmLast] OF FB_SetAlarm;

	  	Alm_bHMIClearHistory:   BOOL;(*清除历史报警*)
		Alm_bBtReset:			BOOL;//报警清除按钮
	  	Alm_iHMIAlarmID:       	DINT;(*当前报警id,给循环显示用*)
		tActSystemTime: 		TIMESTRUCT;//当前系统时间
		gwsActEventMsg:			WSTRING(255);//当前显示的报警信息，跑马灯形式
		gsWriteToLog:			STRING(255);//当前需要添加到报警历史文件的信息
		CurrentLanguage:		STRING;
		
END_VAR

VAR_GLOBAL PERSISTENT(*断电保存型变量,历史报警*)
	   	AlarmHistoryArray :		ARRAY [cnAlmHistoryFirst..cnAlmHistoryLast] OF Alm_AlarmHistoryType;(*记录历史警报状态的数组*)
END_VAR

(*
-------------------------------------在调用的程序里请定义如下变量:----------------------------------------------
*)
VAR_GLOBAL CONSTANT
		cnAlarmFirst:                             	DINT:=1;(*报警的最小id号，默认为1，不需改动*)
		cnAlarmLast:                             	DINT:=1000;(*报警的最大id号*)
		cnAlmActiveFirst:                       	DINT:=1;(*当前激活的警报最小id号，默认为1，不需改动*)
		cnAlmActiveLast:                       		DINT:=1000;(*当前激活的警报最大id号*)
		cnAlmHistoryFirst:                    		DINT:=1;(*历史警报最小id号，默认为1，不需改动*)
		cnAlmHistoryLast:                   	 	DINT:=1000;(*历史警报最大id号*)
END_VAR

// ---- POUs/002_Modbus/BackPrg/PRG_COMM.TcPOU
(***************背景程序，需快速扫描周期********************)
PROGRAM PRG_COMM
VAR
END_VAR


(******************液位********************)
COMCONTROL1(                                 //
	Mode:=SERIALLINEMODE_KL6_22B_STANDARD,   //选择硬件类型
	pComIn:= ADR(COMIN1),                     // pointer to the input variables of the process data of 
                                              //the serial terminal
	pComOut:= ADR(COMOUT1),   //串行硬件进程数据输入变量的通用指针
                              //(数据类型为KL6inData、KL6inData5b、KL6inData22b、EL6inData22b、PcComInData)。
                              //指针是用ADR()函数指定的。
	SizeComIn:= SIZEOF(COMIN1),//正在使用的串行硬件的输入进程映像的大小。大小由SIZEOF()函数确定并分配
	TxBuffer:=TXBUFFER1 ,                    //发送缓存
	RxBuffer:= RXBUFFER1,                    //接收缓存
	Error=> ,
	ErrorID=> );
(******************UVLed********************)	
COMCONTROL2(                                 //
	Mode:=SERIALLINEMODE_KL6_22B_STANDARD,
	pComIn:= ADR(COMIN2),                                                                  
	pComOut:= ADR(COMOUT2),                                                         
	SizeComIn:= SIZEOF(COMIN2),
	TxBuffer:=TXBUFFER2 ,                    
	RxBuffer:= RXBUFFER2,                    
	Error=> ,
	ErrorID=> );

END_PROGRAM

// ---- POUs/000_程序辅助系统/报警/Alarm_FB/FB_AlarmMain.TcPOU
FUNCTION_BLOCK FB_AlarmMAIN(*报警主功能块,请调用一次*)
VAR_INPUT
END_VAR
VAR_OUTPUT
	EventId:			DINT;(*报警号.有报警时会轮询输出有报警的id号*)
   	EventMessage:       WSTRING(255);(*报警信息.有报警时会轮询输出有报警的id信息*)
	EventAlive:			BOOL;(*当前有报警*)
	EventClass:			Alm_EventClass;(*当前的最大报警等级*)
  	NoStopAlarm:        BOOL;(*有小于7的报警,不停机报警*)
   	StopAlarm:          BOOL;(*有大于6的报警,停机报警*)
   	ShowlampOn:         BOOL;(*报警灯亮*)
   	FalshLamp:          BOOL;(*报警灯闪亮.有报警时该信号闪烁输出*)

	AutoRunOff:			BOOL;(*退出自动循环*)
	AlarmAction1:		BOOL;(*用户定义报警动作*)(*例如定义为黄灯亮,则有报警号有触发时,该输出信号为1*)
	AlarmAction2:		BOOL;(*用户定义报警动作*)
	AlarmAction3:		BOOL;(*用户定义报警动作*)
	AlarmAction4:		BOOL;(*用户定义报警动作*)
	AlarmAction5:		BOOL;(*用户定义报警动作*)
	AlarmAction6:		BOOL;(*用户定义报警动作*)
	AlarmAction7:		BOOL;(*用户定义报警动作*)
	AlarmAction8:		BOOL;(*用户定义报警动作*)
END_VAR
VAR
	nConut:                          DINT;
   	fbFreePluse:                     TON;
	m:                               DINT;
	Resul:                           DINT;
	n:                               DINT;
	R_TRIG_AlarmShow:        		 R_TRIG;
	R_TRIG_AlarmAlive:          	 R_TRIG;
	FB_FreePluse_AlarmShow: 		 TON;
	FB_FreePluse_AlarmAlive: 		 TON;
	F_TRIG_bHMIClearHistory: 		 F_TRIG;
	F_TRIG_EventAlive: 				 F_TRIG;
	InstLocalSystemTime:			 FB_LocalSystemTime;
END_VAR

(*Set Signal*)
 	EventAlive:=ShowlampOn:=AlarmAction1:=AlarmAction2:=AlarmAction3:=FALSE;
  	AlarmAction4:=AlarmAction5:=AlarmAction6:=AlarmAction7:=AlarmAction8:=FALSE;
	AutoRunOff :=	FALSE;(*退出自动循环*)
   	EventClass :=	0;

FOR nConut :=cnAlarmFirst TO cnAlarmLast DO
	    EventAlive :=	EventAlive OR AlarmActionArray[nConut].EventAlive;
	    ShowlampOn :=	ShowlampOn OR AlarmActionArray[nConut].ShowlampOn;
	    AlarmAction1:=	AlarmAction1 OR AlarmActionArray[nConut].AlarmAction1;
	    AlarmAction2:=	AlarmAction2 OR AlarmActionArray[nConut].AlarmAction2;
	    AlarmAction3:=	AlarmAction3 OR AlarmActionArray[nConut].AlarmAction3;
	    AlarmAction4:=	AlarmAction4 OR AlarmActionArray[nConut].AlarmAction4;
	    AlarmAction5:=	AlarmAction5 OR AlarmActionArray[nConut].AlarmAction5;
	    AlarmAction6:=	AlarmAction6 OR AlarmActionArray[nConut].AlarmAction6;
	    AlarmAction7:=	AlarmAction7 OR AlarmActionArray[nConut].AlarmAction7;
	    AlarmAction8:=	AlarmAction8 OR AlarmActionArray[nConut].AlarmAction8;
	    AutoRunOff :=	AutoRunOff 	OR AlarmActionArray[nConut].AutoRunOff;
	    EventClass  :=	MAX(EventClass,AlarmActionArray[nConut].EventClass);
END_FOR

(*Flash lamp*)
R_TRIG_AlarmShow(CLK:=ShowlampOn  );
IF ShowlampOn THEN              (****有报警时，先初始化时间输入为FALSE，灯亮，然后开始下步TON运行1S，闪灯状态变化
                                      优点：一有报警，就灯亮，避免有报警时过1S灯才亮*)
	IF R_TRIG_AlarmShow.Q THEN
		fbFreePluse(IN:=FALSE);
		FalshLamp:=TRUE;
	END_IF
	fbFreePluse(IN:=NOT fbFreePluse.Q,PT:=T#1S);
	IF fbFreePluse.Q THEN
		FalshLamp:=NOT FalshLamp;
	END_IF
ELSE
	FalshLamp:=FALSE;
END_IF



(*Action*)
AlarmAlive();
AlarmHMI();
AlarmShow();

(*Set Action*)
IF EventAlive THEN
     IF EventClass>6 THEN
         StopAlarm:=TRUE;
         NoStopAlarm:=FALSE;
     ELSE
         StopAlarm:=FALSE;
         NoStopAlarm:=TRUE;
    END_IF
ELSE
    StopAlarm:=FALSE;
    NoStopAlarm:=FALSE;
    EventId:=0;
    EventMessage:="";
    Alm_iHMIAlarmID:=0;
END_IF

	//获取系统时间
	InstLocalSystemTime(
		sNetID		:= '',
		bEnable		:= TRUE,
		dwCycle		:= 1,
		systemTime	=> tActSystemTime,
		);

ACTION AlarmAlive:
(*总报警数有n个，用其中有报警的[2],[4]赋值给激活报警m[1],[2],m自加1，然后循环比较m-20,把信息格式化*)
(*-----------------------------------当前报警列表显示-----------------------------*)
R_TRIG_AlarmAlive(CLK:=EventAlive);
IF EventAlive THEN
	IF R_TRIG_AlarmAlive.Q THEN
   	 	FB_FreePluse_AlarmAlive(In:=FALSE);
	END_IF
    FB_FreePluse_AlarmAlive(In:= NOT FB_FreePluse_AlarmAlive.Q,PT:=T#1S );
    IF FB_FreePluse_AlarmAlive.Q OR R_TRIG_AlarmAlive.Q THEN
         n:=cnAlarmFirst;
         m:=cnAlmActiveFirst;
          FOR n:=cnAlarmFirst TO cnAlarmLast DO     (*把所有报警赋值到当前激活报警数组*)
               IF AlarmActionArray[n].EventAlive THEN
                    AlarmActiveArray[m].EventId       :=AlarmActionArray[n].EventId;
                   	AlarmActiveArray[m].EventMessage  :=AlarmActionArray[n].EventMessage;						
                    AlarmActiveArray[m].EventTime     :=AlarmActionArray[n].EventTime;
                  	m:=m+1;
                    IF m>cnAlmActiveLast THEN
                       n:=32766;  (*exit FOR*)
                    END_IF
               END_IF
         END_FOR
         IF m<cnAlmActiveLast THEN
               FOR n:=m TO cnAlmActiveLast DO
                   AlarmActiveArray[n].EventId:=0;
                 	AlarmActiveArray[n].EventMessage:="";
                   	AlarmActiveArray[n].EventTime:=DT#2000-01-01-00:00;
             END_FOR
          END_IF
    END_IF
END_IF
(*当报警消失时,把显示列表内容清空*)
F_TRIG_EventAlive(CLK:=EventAlive );
IF F_TRIG_EventAlive.Q THEN
	FOR n:=cnAlmActiveFirst TO cnAlmActiveLast DO 
		AlarmActiveArray[n].EventId:=0;
		AlarmActiveArray[n].EventMessage:="";
		AlarmActiveArray[n].EventTime:=DT#2016-01-01-00:00;
	END_FOR
END_IF
END_ACTION

ACTION AlarmHMI:


(*``````````````````````````````````````````清除历史报警`````````````````````````````````````*)
F_TRIG_bHMIClearHistory(CLK:=Alm_bHMIClearHistory  );
IF F_TRIG_bHMIClearHistory.Q THEN
       FOR n:=cnAlmHistoryFirst TO cnAlmHistoryLast DO
             AlarmHistoryArray[n].EventId:=0;
             AlarmHistoryArray[n].EventMessage:="";
             AlarmHistoryArray[n].EventTime:=DT#2016-01-01-00:00;
        END_FOR
        Alm_HistoryAlarmNum:=0;
END_IF
END_ACTION

ACTION AlarmShow:

(*-------------------------------跑马灯显示报警---------------------------------*)
FB_FreePluse_AlarmShow(IN:=NOT FB_FreePluse_AlarmShow.Q,PT:=T#1S );
IF FB_FreePluse_AlarmShow.Q OR R_TRIG_AlarmAlive.Q THEN
      n:=EventId;
      	FOR m:=n+1 TO cnAlarmLast DO
            IF AlarmActionArray[m].EventAlive THEN
                   n:=m;
                   m:=cnAlarmLast+10;
             END_IF;
      	END_FOR;
    	IF n<>EventId THEN
        	Resul:=n;     
   		ELSE
          	FOR m:=cnAlarmFirst TO cnAlarmLast DO
             	IF AlarmActionArray[m].EventAlive THEN
                 	n:=m;
                 	m:=cnAlarmLast+10;
              	END_IF;
          	END_FOR;
          	Resul:=n;
      	END_IF
END_IF

Alm_iHMIAlarmID:=EventId:=Resul;
IF EventId<=cnAlarmLast AND EventId>= cnAlarmFirst THEN
	gwsActEventMsg:=EventMessage:=AlarmActionArray[EventId].EventMessage;
ELSE
	gwsActEventMsg:=EventMessage:="";	
END_IF
END_ACTION

END_FUNCTION_BLOCK

// ---- POUs/000_程序辅助系统/报警/Alarm_FB/Products/FB_FileCopy.TcPOU
FUNCTION_BLOCK FB_FileCopy
VAR_INPUT
	srcNetId				: T_AmsNetId;	(* TwinCAT network address of the source file *)
	srcFileName			: T_MaxString;	(* source file path and name *)
	destNetId			: T_AmsNetId;	(* TwinCAT network address of the destination file *)
	destFileName		: T_MaxString;  (* destination file path and name *)
	bExecute			: BOOL;			(* rising edge start fb execution *)
	tAdsTimeOut			: TIME;			(* ads timeout *)
	cbReadLen			: UDINT;
END_VAR
VAR_OUTPUT
	bBusy				:BOOL;
	bError				:BOOL;
	nErrId				:UDINT;
END_VAR
VAR
	fbFileOpen			:FB_FileOpen;
	fbFileClose			:FB_FileClose;
	fbFileRead			:FB_FileRead;
	fbFileWrite			:FB_FileWrite;

	hSrcFile				:UINT	:= 0;(* file handle of the source file *)
	hDestFile			:UINT	:= 0;(* file handle of the destination file *)

	Step				:DWORD;
	RisingEdge			:R_TRIG;

	buffRead				:ARRAY[1..30000] OF BYTE;(* buffer *)
	cbReadLength		:UDINT:=0;
	TimeCount			:INT;
END_VAR

RisingEdge(CLK:=bExecute);
IF RisingEdge.Q THEN
	IF NOT bBusy THEN
		bBusy := TRUE;
		bError:= FALSE;
		nErrId:=0;
		Step := 1;
		cbReadLength:=0;
		hSrcFile:=0;
		hDestFile:=0;
		TimeCount:=0;
	END_IF
END_IF

IF bBusy THEN
	TimeCount:=TimeCount+1;
END_IF


CASE Step OF
	0:	(* do nothing *)
		;

	1:	(* open source file *)
		fbFileOpen(  bExecute := FALSE  );
		fbFileOpen( 	sNetId := srcNetId,
						sPathName := srcFileName,
						nMode := FOPEN_MODEREAD OR FOPEN_MODEBINARY(*FOPEN_MODETEXT*),
						ePath := PATH_GENERIC,
						tTimeout := tAdsTimeout,
						bExecute := TRUE );
		Step := Step + 1;

	2:
		fbFileOpen( bExecute := FALSE );
		IF ( NOT fbFileOpen.bBusy ) THEN
			IF ( fbFileOpen.bError ) THEN
				nErrId := fbFileOpen.nErrId;
				bError := TRUE;
				Step := 50;
			ELSE
				hSrcFile := fbFileOpen.hFile;
				Step := Step + 1;
			END_IF
		END_IF

	3:	(* open destination file *)
		fbFileOpen(  bExecute := FALSE  );
		fbFileOpen( 	sNetId := destNetId,
						sPathName := destFileName,
						nMode := FOPEN_MODEWRITE OR FOPEN_MODEBINARY(*FOPEN_MODETEXT*),
						ePath := PATH_GENERIC,
						tTimeout := tAdsTimeout,
						bExecute := TRUE );
		Step := Step+1;

	4:
		fbFileOpen(  bExecute := FALSE  );
		IF ( NOT fbFileOpen.bBusy ) THEN
			IF ( fbFileOpen.bError ) THEN
				nErrId := fbFileOpen.nErrId;
				bError := TRUE;
				Step := 50;
			ELSE
				hDestFile := fbFileOpen.hFile;
				Step := Step + 1;
			END_IF
		END_IF

	5:	(*read data from source file*)
		cbReadLength := 0;
		fbFileRead( bExecute:= FALSE );
		fbFileRead( 	sNetId:=SrcNetId,
						hFile:=hSrcFile,
						pReadBuff:= ADR(buffRead),
						cbReadLen:= (*SIZEOF(buffRead)*)cbReadLen,
						bExecute:=TRUE,
						tTimeout:=tAdsTimeOut );
		Step := Step + 1;

	6:
		fbFileRead( bExecute:= FALSE );
		IF ( NOT fbFileRead.bBusy ) THEN
			IF ( fbFileRead.bError ) THEN
				nErrId := fbFileRead.nErrId;
				bError := TRUE;
				Step := 50;
			ELSE
				cbReadLength := fbFileRead.cbRead;
				Step := Step + 1;
			END_IF
		END_IF

	7:	(*write data to destination file*)
		fbFileWrite( bExecute := FALSE );
		fbFileWrite(	sNetId:=DestNetId,
						hFile:=hDestFile,
						pWriteBuff:= ADR(buffRead),
						cbWriteLen:= cbReadLength,
						bExecute:=TRUE,
						tTimeout:=tAdsTimeOut );
		Step := Step + 1;

	8:
		fbFileWrite( bExecute := FALSE );
		IF ( NOT fbFileWrite.bBusy ) THEN
			IF ( fbFileWrite.bError ) THEN
				nErrId := fbFileWrite.nErrId;
				bError := TRUE;
				Step := 50;
			ELSE
				IF fbFileRead.bEOF THEN (*Check if the EOF flag ist set *)
					Step := 50;		(*cleanup: close the destination and source files *)
				ELSE
					Step := 5; (* repeat reading *)
				END_IF
			END_IF
		END_IF

	30:	(* close the destination file *)
		fbFileClose( bExecute := FALSE );
		fbFileClose( 	sNetId:=destNetId,
						hFile:=hDestFile,
						bExecute:=TRUE,
						tTimeout:=tAdsTimeOut );
		Step := Step + 1;

	31:
		fbFileClose( bExecute := FALSE );
		IF ( NOT fbFileClose.bBusy ) THEN
			IF ( fbFileClose.bError ) THEN
				nErrId := fbFileClose.nErrId;
				bError := TRUE;
			END_IF
			Step := 50;
			hDestFile := 0;
		END_IF

	40: (* close source file *)
		fbFileClose( bExecute := FALSE );
		fbFileClose( 	sNetId:=srcNetId,
						hFile:=hSrcFile,
						bExecute:=TRUE,
						tTimeout:=tAdsTimeOut );
		Step := Step + 1;

	41:
		fbFileClose( bExecute := FALSE );
		IF ( NOT fbFileClose.bBusy ) THEN
			IF ( fbFileClose.bError ) THEN
				nErrId := fbFileClose.nErrId;
				bError := TRUE;
			END_IF
			Step := 50;
			hSrcFile := 0;
		END_IF

	50: (*error or ready => cleanup*)
		IF ( hDestFile <> 0 ) THEN
			Step := 30; (* close the destination file*)
		ELSIF (hSrcFile <> 0 ) THEN
			Step := 40; (* close the source file *)
		ELSE
			Step := 0;	(* ready *)
			bBusy := FALSE;
		END_IF

END_CASE

END_FUNCTION_BLOCK

// ---- POUs/000_程序辅助系统/报警/Alarm_FB/SW_FormatWstring.TcPOU
FUNCTION_BLOCK SW_FormatWstring//格式化字符串
VAR_INPUT
	WstringIn:			WSTRING(255);
	D1:					DINT;
	D2:					DINT;
	S1:					STRING(255);
END_VAR
VAR_OUTPUT
	WstringOUT:			WSTRING(255);
END_VAR
VAR
	Var1: 				INT;
END_VAR


Var1:=WFIND(WstringIn,"%D");
IF Var1<>0 THEN
	WstringOUT := WREPLACE(WstringIn,DINT_TO_WSTRING(D1),2,Var1);

	Var1:=WFIND(WstringOUT,"%D");
	IF Var1<>0 THEN
		WstringOUT := WREPLACE(WstringOUT,DINT_TO_WSTRING(D2),2,Var1);
	END_IF
ELSE
	WstringOUT:=WstringIN;
END_IF

Var1:=WFIND(WstringOUT,"%S");
IF Var1<>0 THEN
	WstringOUT := WREPLACE(WstringOUT,STRING_TO_WSTRING(S1),2,Var1);
END_IF

END_FUNCTION_BLOCK

// ---- POUs/000_程序辅助系统/系统功能/systime.TcPOU
PROGRAM systime
VAR
	fb_localsystime1:Tc2_Utilities.FB_LocalSystemTime;
	systime1:Tc2_Utilities.TIMESTRUCT;
	dttime:DATE_AND_TIME;
	todacttime:TIME_OF_DAY;
	sTime,sData	:STRING;
END_VAR

fb_localsystime1(
	sNetID:= , 
	bEnable:= TRUE, 
	dwCycle:= , 
	dwOpt:= , 
	tTimeout:= , 
	bValid=> , 
	systemTime=>systime1 , 
	tzID=> );
	
dttime:=Tc2_Utilities.SYSTEMTIME_TO_DT(systime1);
todacttime:=DT_TO_TOD(dttime);
    sTime := concat(WORD_TO_STRING(fb_localsystime1.systemTime.wHour),':');
	sTime := concat(sTime,WORD_TO_STRING(fb_localsystime1.systemTime.wMinute));
	sTime := concat(sTime,':');
	sTime := concat(sTime,WORD_TO_STRING(fb_localsystime1.systemTime.wSecond));
(*	sData := concat(WORD_TO_STRING(fb_localsystime1.systemTime.wDayOfWeek),',');
	sData := Tc2_Standard.CONCAT(sData,WORD_TO_STRING(fb_localsystime1.systemTime.wMonth));
	sData := Tc2_Standard.CONCAT(sdata,'.');
	sData := Tc2_Standard.CONCAT(sData,WORD_TO_STRING(fb_localsystime1.systemTime.wDay));
	sData := Tc2_Standard.CONCAT(sData,',');
	sData := Tc2_Standard.CONCAT(sData,WORD_TO_STRING(fb_localsystime1.systemTime.wYear));
	*)

END_PROGRAM

// ---- POUs/001_FB/FB_Buzzer.TcPOU
FUNCTION_BLOCK FB_Buzzer
VAR_INPUT	
	duration:LREAL;//S,总时间
	period :LREAL;//S,周期时间
END_VAR
VAR_OUTPUT
	bqbuzzer:BOOL;
END_VAR
VAR
		ton1,ton2       :Tc2_Standard.TON;
		en_trig:R_TRIG;
		ton_duration:TON;
		enable:BOOL;
END_VAR
VAR_IN_OUT
	Start_Exe:BOOL;
END_VAR

en_trig(CLK:=Start_Exe , Q=> );
IF en_trig.Q THEN 
	enable:=TRUE;
	bqbuzzer:=TRUE;
END_IF
IF NOT Start_Exe THEN 
	enable:=FALSE;
END_IF

IF enable THEN 
	ton1(IN:= bqbuzzer, PT:= LREAL_TO_TIME(period)*1000, Q=> , ET=> );
	ton2(IN:= NOT bqbuzzer, PT:=LREAL_TO_TIME(period)*1000 , Q=> , ET=> );
	ton_duration(IN:=TRUE , PT:=LREAL_TO_TIME(duration)*1000 , Q=> , ET=> );
	IF ton1.Q OR ton2.Q THEN
		bqbuzzer:=NOT bqbuzzer;
	END_IF
	IF ton_duration.Q THEN 
		enable:=FALSE;
		Start_Exe:=FALSE;
	END_IF
ELSE 
	bqbuzzer:=FALSE;
	ton1(IN:=FALSE);
	ton2(IN:=FALSE);
	ton_duration(IN:=FALSE);
END_IF

END_FUNCTION_BLOCK

// ---- POUs/001_FB/FB_SQUARE.TcPOU
FUNCTION_BLOCK FB_SQUARE
VAR_INPUT
	T_ON	:LREAL;//s
	T_OFF	:LREAL;//s
END_VAR
VAR_OUTPUT
	SQUARE:BOOL;
END_VAR
VAR
	Ton1,Ton2:TON;
	step:INT;
END_VAR

ton1(IN:=NOT SQUARE, PT:= LREAL_TO_TIME(T_OFF*1000), Q=> , ET=> );
ton2(IN:=  SQUARE, PT:=LREAL_TO_TIME(T_ON*1000) , Q=> , ET=> );
IF ton1.Q OR ton2.Q THEN
	SQUARE:=NOT SQUARE;
END_IF

END_FUNCTION_BLOCK

// ---- POUs/002_Modbus/P_Modbus.TcPOU
PROGRAM P_Modbus
VAR
END_VAR

P_Modbus_RTU();
PRG_SerialComm();

END_PROGRAM

// ---- POUs/003_Input_Output/IO_Link.TcPOU
PROGRAM IO_Link
VAR

	test: BOOL;
END_VAR

Act_Inputs();
Act_Outputs();

GVL_API.stInput:=stInput;
GVL_API.stOutput:=stOutput;
GVL_API.Axis_SpitUnit_snHome    :=Axis[SpitUnit].	IO.snHome;
GVL_API.Axis_SpitUnit_snLimitP  :=Axis[SpitUnit].	IO.snLimitP;

ACTION Act_Inputs:
(**DI1**)
Axis[FastScan].IO.snHome	(*	Fast Scan 原点	*)	:=	EL1809_M[1	,1]	;
Axis[SpitUnit].	IO.snHome	(*	闪喷糟原点	*)	:=	EL1809_M[1	,2]	;
Axis[SpitUnit].	IO.snLimitP	(*	闪喷糟极限	*)	:=	EL1809_M[1	,3]	;
stInput.	biUDS_sensor_up_S[1]	(*	压辊S1上限位	*)	:=	EL1809_M[1	,4]	;
stInput.	biUDS_sensor_up_S[2]	(*	压辊S2上限位	*)	:=	EL1809_M[1	,5]	;
stInput.	biUDS_sensor_up_S[3]	(*	压辊S3上限位	*)	:=	EL1809_M[1	,6]	;
stInput.	biUDS_sensor_up_S[4]	(*	压辊S4上限位	*)	:=	EL1809_M[1	,7]	;
stInput.	biUDS_sensor_up_S[5]	(*	压辊S5上限位	*)	:=	EL1809_M[1	,8]	;
stInput.	biUDS_sensor_up_S[6]	(*	压辊S6上限位	*)	:=	EL1809_M[1	,9]	;
stInput.	biUDS_sensor_down_S1[1]	(*	压辊S1下限位1	*)	:=	EL1809_M[1	,10]	;
stInput.	biUDS_sensor_down_S1[2]	(*	压辊S1下限位2	*)	:=	EL1809_M[1	,11]	;
stInput.	biUDS_sensor_down_S1[3]	(*	压辊S1下限位3	*)	:=	EL1809_M[1	,12]	;
stInput.	biUDS_sensor_down_S1[4]	(*	压辊S1下限位4	*)	:=	EL1809_M[1	,13]	;
stInput.	biUDS_sensor_down_S1[5]	(*	压辊S1下限位5	*)	:=	EL1809_M[1	,14]	;
stInput.	biUDS_sensor_down_S1[6]	(*	压辊S1下限位6	*)	:=	EL1809_M[1	,15]	;
stInput.	biUDS_sensor_down_S1[7]	(*	压辊S1下限位7	*)	:=	EL1809_M[1	,16]	;

(**DI2**)
stInput.	biUDS_sensor_down_S1[8]	(*	压辊S1下限位8	*)	:=	EL1809_M[2	,1]	;
stInput.	biUDS_sensor_down_S1[9]	(*	压辊S1下限位9	*)	:=	EL1809_M[2	,2]	;
stInput.	biUDS_sensor_down_S1[10]	(*	压辊S1下限位10	*)	:=	EL1809_M[2	,3]	;
stInput.	biUDS_sensor_down_S1[11]	(*	压辊S1下限位11	*)	:=	EL1809_M[2	,4]	;
stInput.	biUDS_sensor_down_S1[12]	(*	压辊S1下限位12	*)	:=	EL1809_M[2	,5]	;
stInput.	biUDS_sensor_down_S1[13]	(*	压辊S1下限位13	*)	:=	EL1809_M[2	,6]	;
stInput.	biUDS_sensor_down_S1[14]	(*	压辊S1下限位14	*)	:=	EL1809_M[2	,7]	;
stInput.	biUDS_sensor_down_S1[15]	(*	压辊S1下限位15	*)	:=	EL1809_M[2	,8]	;
stInput.	biUDS_sensor_down_S1[16]	(*	压辊S1下限位16	*)	:=	EL1809_M[2	,9]	;
stInput.	biFootPedal[1].PedalPressed1	(*	左前脚踏开关1	*)	:=	EL1809_M[2	,10]	;
stInput.	biFootPedal[1].PedalPressed2	(*	左前脚踏开关2	*)	:=	EL1809_M[2	,11]	;
stInput.	biFootPedal[1].PedalPressed3	(*	左前脚踏开关3	*)	:=	EL1809_M[2	,12]	;
stInput.	biFootPedal[3].PedalPressed1	(*	右前脚踏开关1	*)	:=	EL1809_M[2	,13]	;
stInput.	biFootPedal[3].PedalPressed2	(*	右前脚踏开关2	*)	:=	EL1809_M[2	,14]	;
stInput.	biFootPedal[3].PedalPressed3	(*	右前脚踏开关3	*)	:=	EL1809_M[2	,15]	;
stInput.	biFootPedal[2].PedalPressed1	(*	左后脚踏开关1	*)	:=	EL1809_M[2	,16]	;

(**DI3**)
stInput.	biFootPedal[2].PedalPressed2	(*	左后脚踏开关2	*)	:=	EL1809_M[3	,1]	;
stInput.	biFootPedal[2].PedalPressed3	(*	左后脚踏开关3	*)	:=	EL1809_M[3	,2]	;
stInput.	biFootPedal[4].PedalPressed1	(*	右后脚踏开关1	*)	:=	EL1809_M[3	,3]	;
stInput.	biFootPedal[4].PedalPressed2	(*	右后脚踏开关2	*)	:=	EL1809_M[3	,4]	;
stInput.	biFootPedal[4].PedalPressed3	(*	右后脚踏开关3	*)	:=	EL1809_M[3	,5]	;
stInput.	biDualSensor[1]	(*	单/双roll检测限位input	*)	:=	EL1809_M[3	,6]	;
stInput.	biDualSensor[2]	(*	单/双roll检测限位output	*)	:=	EL1809_M[3	,7]	;
stInput.	biClamp_hold[1]	(*	卡盘到位检测input	*)	:=	EL1809_M[3	,8]	;
stInput.	biClamp_hold[2]	(*	卡盘到位检测output	*)	:=	EL1809_M[3	,9]	;

(**SDI1**)
stInput.	biElectromagnet_limit	(*	探块限位	*)	:=	EL1809_S[1	,1]	;
Axis[Z_Axis].	IO.snHome	(*	Z轴原点	*)	:=	EL1809_S[1	,2]	;
Axis[Z_Axis].	IO.snLimitP	(*	Z轴下极限	*)	:=	EL1809_S[1	,3]	;
stInput.	biSubInkTankLevel[9]	(*	二级墨盒液位C1	*)	:=	NOT	EL1809_S[1	,4]	;
stInput.	biSubInkTankLevel[10]	(*	二级墨盒液位C2	*)	:=	NOT	EL1809_S[1	,5]	;
stInput.	biSubInkTankLevel[5]	(*	二级墨盒液位Y1	*)	:=	NOT	EL1809_S[1	,6]	;
stInput.	biSubInkTankLevel[6]	(*	二级墨盒液位Y2	*)	:=	NOT	EL1809_S[1	,7]	;
stInput.	biSubInkTankLevel[7]	(*	二级墨盒液位M1	*)	:=	NOT	EL1809_S[1	,8]	;
stInput.	biSubInkTankLevel[8]	(*	二级墨盒液位M2	*)	:=	NOT	EL1809_S[1	,9]	;
stInput.	biSubInkTankLevel[11]	(*	二级墨盒液位K1	*)	:=	NOT	EL1809_S[1	,10]	;
stInput.	biSubInkTankLevel[12]	(*	二级墨盒液位K2	*)	:=	NOT	EL1809_S[1	,11]	;
stInput.	biSubInkTankLevel[1]	(*	二级墨盒液位LC1	*)	:=	NOT	EL1809_S[1	,12]	;
stInput.	biSubInkTankLevel[2]	(*	二级墨盒液位LC2	*)	:=	NOT	EL1809_S[1	,13]	;
stInput.	biSubInkTankLevel[3]	(*	二级墨盒液位LM1	*)	:=	NOT	EL1809_S[1	,14]	;
stInput.	biSubInkTankLevel[4]	(*	二级墨盒液位LM2	*)	:=	NOT	EL1809_S[1	,15]	;
stInput.	biSubInkTankLevel[17]	(*	二级墨盒液位图层1	*)	:=	NOT	EL1809_S[1	,16]	;


(**SDI2**)
stInput.	biSubInkTankLevel[18]	(*	二级墨盒液位图层2	*)	:=	NOT	EL1809_S[2	,1]	;
stInput.	biSubInkTankLevel[13]	(*	二级墨盒液位W1	*)	:=	NOT	EL1809_S[2	,2]	;
stInput.	biSubInkTankLevel[14]	(*	二级墨盒液位W2	*)	:=	NOT	EL1809_S[2	,3]	;
stInput.	biSubInkTankLevel[15]	(*	二级墨盒液位W3	*)	:=	NOT	EL1809_S[2	,4]	;
stInput.	biSubInkTankLevel[16]	(*	二级墨盒液位W4	*)	:=	NOT	EL1809_S[2	,5]	;


stInput.	biProtectAirTankLevel_C	(*	真空保护瓶液位_彩	*)	:=	EL1809_S[2	,6]	;
stInput.	biProtectAirTankLevel_W	(*	真空保护瓶液位_白	*)	:=	EL1809_S[2	,7]	;
stInput.	btPurge	(*	正压按钮	*)	:=	EL1809_S[2	,8]	;
stInput.	btVacBt_C	(*	彩色正负压切换按钮	*)	:=	EL1809_S[2	,9]	;
stInput.	btVacBt_W	(*	白色正负压切换按钮	*)	:=	EL1809_S[2	,10]	;


(***************************Main Ink Tank****************)

	
(***************************Sub Ink Tank******************)
END_ACTION

ACTION Act_Outputs:

(**DO1**)
EL2809_M[1	,1]	:=	stOutput.	bqFillPumpWorking[19]	;	(*	清洗液泵1	*)
EL2809_M[1	,2]	:=	stOutput.	bqFillPumpWorking[20]	;	(*	清洗液泵2	*)
EL2809_M[1	,3]	:=	stOutput.	bqStirrerWorkingF	;	(*	白墨瓶搅拌（正转）	*)
EL2809_M[1	,4]	:=	stOutput.	bqStirrerWorkingB	;	(*	白墨瓶搅拌（反转）	*)
EL2809_M[1	,5]	:=	stOutput.	bqsensor_blink[5]	;	(*	墨瓶C  LED	*)
EL2809_M[1	,6]	:=	stOutput.	bqsensor_blink[3]	;	(*	墨瓶Y  LED	*)
EL2809_M[1	,7]	:=	stOutput.	bqsensor_blink[4]	;	(*	墨瓶M  LED	*)
EL2809_M[1	,8]	:=	stOutput.	bqsensor_blink[6]	;	(*	墨瓶K  LED	*)
EL2809_M[1	,9]	:=	stOutput.	bqsensor_blink[1]	;	(*	墨瓶LC  LED	*)
EL2809_M[1	,10]	:=	stOutput.	bqsensor_blink[2]	;	(*	墨瓶LM  LED	*)
EL2809_M[1	,11]	:=	stOutput.	bqsensor_blink[9]	;	(*	墨瓶图层  LED	*)
EL2809_M[1	,12]	:=	stOutput.	bqsensor_blink[7]	;	(*	墨瓶W  LED	*)
EL2809_M[1	,13]	:=	stOutput.	bqsensor_blink[8]	;	(*	墨瓶清洗液  LED	*)
EL2809_M[1	,14]	:=	stOutput.	bqsensor_blink[10]	;	(*	墨瓶废液  LED	*)
EL2809_M[1	,15]	:=	stOutput.	bqFanPower	;	(*	废液吸风扇	*)
EL2809_M[1	,16]	:=	stOutput.	bqWastePump	;	(*	废液泵	*)

(**DO2**)
EL2809_M[2	,1]	:=	stOutput.	bqBreakPower[1]	;		(*	放卷L_刹车	*)
EL2809_M[2	,2]	:=	stOutput.	bqCluthOut[1]	;		(*	放卷L_离合器out	*)
EL2809_M[2	,3]	:=	stOutput.	bqReset[1]	;		(*	放卷L_离合器rst	*)
EL2809_M[2	,4]	:=	stOutput.	bqBreakPower[3]	;		(*	放卷R_刹车	*)
EL2809_M[2	,5]	:=	stOutput.	bqCluthOut[3]	;		(*	放卷R_离合器out	*)
EL2809_M[2	,6]	:=	stOutput.	bqReset[3]	;		(*	放卷R_离合器rst	*)
EL2809_M[2	,7]	:=	stOutput.	bqCluthOut[2]	;		(*	收卷L_离合器out	*)
EL2809_M[2	,8]	:=	stOutput.	bqReset[2]	;		(*	收卷L_离合器rst	*)
EL2809_M[2	,9]	:=	stOutput.	bqCluthOut[4]	;		(*	收卷R_离合器out	*)
EL2809_M[2	,10]	:=	stOutput.	bqReset[4]	;		(*	收卷R_离合器rst	*)
EL2809_M[2	,11]	:=	stOutput.	bqS1_Drive_enabled	;	(*	导向压轮电机使能	*)
EL2809_M[2	,12]	:=	stOutput.	bqS1_Forward_Reverse	;	(*	导向压轮电机正/反转	*)
EL2809_M[2	,13]	:=	stOutput.	bqS1_Break	;	(*	导向压轮电机刹车	*)

(**DO3**)
EL2809_M[3	,1]	:=	stOutput.	bqVacRun[1]	;	(*	真空吸附启停	*)
EL2809_M[3	,2]	:=	stOutput.	bqUDS_MoveUp_do[2]	;		(*	压辊气缸S2上升	*)
EL2809_M[3	,3]	:=	stOutput.	bqUDS_MoveDown_do[2]	;		(*	压辊气缸S2下降	*)
EL2809_M[3	,4]	:=	stOutput.	bqUDS_MoveUp_do[3]	;		(*	压辊气缸S3上升	*)
EL2809_M[3	,5]	:=	stOutput.	bqUDS_MoveDown_do[3]	;		(*	压辊气缸S3下降	*)
EL2809_M[3	,6]	:=	stOutput.	bqUDS_MoveUp_do[4]	;		(*	压辊气缸S4上升	*)
EL2809_M[3	,7]	:=	stOutput.	bqUDS_MoveDown_do[4]	;		(*	压辊气缸S4下降	*)
EL2809_M[3	,8]	:=	stOutput.	bqUDS_MoveUp_do[5]	;		(*	压辊气缸S5上升	*)
EL2809_M[3	,9]	:=	stOutput.	bqUDS_MoveDown_do[5]	;		(*	压辊气缸S5下降	*)
EL2809_M[3	,10]	:=	stOutput.	bqUDS_MoveUp_do[6]	;		(*	压辊气缸S6上升	*)
EL2809_M[3	,11]	:=	stOutput.	bqUDS_MoveDown_do[6]	;		(*	压辊气缸S6下降	*)


(**DO4**)
EL2809_M[4	,1]	:=	stOutput.	bqFillPumpWorking[9]	;		(*	供墨泵C1	*)
EL2809_M[4	,2]	:=	stOutput.	bqFillPumpWorking[10]	;		(*	供墨泵C2	*)
EL2809_M[4	,3]	:=	stOutput.	bqFillPumpWorking[5]	;		(*	供墨泵Y1	*)
EL2809_M[4	,4]	:=	stOutput.	bqFillPumpWorking[6]	;		(*	供墨泵Y2	*)
EL2809_M[4	,5]	:=	stOutput.	bqFillPumpWorking[7]	;		(*	供墨泵M1	*)
EL2809_M[4	,6]	:=	stOutput.	bqFillPumpWorking[8]	;		(*	供墨泵M2	*)
EL2809_M[4	,7]	:=	stOutput.	bqFillPumpWorking[11]	;		(*	供墨泵K1	*)
EL2809_M[4	,8]	:=	stOutput.	bqFillPumpWorking[12]	;		(*	供墨泵K2	*)
EL2809_M[4	,9]	:=	stOutput.	bqFillPumpWorking[1]	;		(*	供墨泵LC1	*)
EL2809_M[4	,10]	:=	stOutput.	bqFillPumpWorking[2]	;		(*	供墨泵LC2	*)
EL2809_M[4	,11]	:=	stOutput.	bqFillPumpWorking[3]	;		(*	供墨泵LM1	*)
EL2809_M[4	,12]	:=	stOutput.	bqFillPumpWorking[4]	;		(*	供墨泵LM2	*)
EL2809_M[4	,13]	:=	stOutput.	bqFillPumpWorking[17]	;		(*	图层泵1	*)
EL2809_M[4	,14]	:=	stOutput.	bqFillPumpWorking[18]	;		(*	图层泵2	*)
EL2809_M[4	,15]	:=	stOutput.	bqFillPumpWorking[13]	;		(*	供墨泵 W1	*)
EL2809_M[4	,16]	:=	stOutput.	bqFillPumpWorking[15]	;		(*	供墨泵 W2	*)


(**DO1**)
EL2809_S[1	,1]	:=	stOutput.	bqSubCircPumpWorking[1]	;	(*	二级墨盒白循环泵1	*)
EL2809_S[1	,2]	:=	stOutput.	bqSubCircPumpWorking[2]	;	(*	二级墨盒白循环泵2	*)
EL2809_S[1	,3]	:=	stOutput.	bqPurValve	;	(*	正压电磁阀	*)
EL2809_S[1	,4]	:=	stOutput.	bqVacValve_W	;	(*	负压电磁阀白	*)
EL2809_S[1	,5]	:=	stOutput.	bqVacValve_C	;	(*	负压电磁阀彩	*)
EL2809_S[1	,6]	:=	stOutput.	bqElectromagnet_power	;	(*	探块电源	*)
END_ACTION

END_PROGRAM

// ---- POUs/010_Motion/XMove/P_FastScan.TcPOU
PROGRAM P_FastScan
VAR
	ID						:INT:=FastScan;
	SysStep:				DINT;	
	HomeStep:				DINT;	
	RestStep				:DINT;
	MoveStep				:DINT;
	HomeDone:               BOOL;
	FB_move:				FB_MoveFS_Exte;
	FB_home:				FB_Home_X;
	ton_commandtimeout		:TON;

	ton1:Tc2_Standard.TON;	//	命令延迟关闭
	Move_Done				:BOOL;
	NOT_Moving_TimeOut		:BOOL;
	parameter_out_of_range	:BOOL;
	actuator_out_of_pos_range:BOOL;
	actuator_out_of_neg_range:BOOL;	
	homeTimeOut				:BOOL;
	SpeedNotReach			:BOOL;	
	jog_EN					:BOOL;
	ton_Moving				:TON;
	
	direN:BOOL;
	direp:BOOL;
	log_ErrorEnum:Axis_XY_ErrorEnum;
	log_ID:INT;
	i:INT;
	
END_VAR

ACT_LOG();
GVL_API.stAxis[ID].ControlLoopClosed:=Axis[ID].Ref.Status .ControlLoopClosed;

(*****************POS******************************)
GVL_API.stAxis[ID].position:=Axis[ID].Ref.NcToPlc.ActPos;
direN:=Axis[ID].Ref.Status.NegativeDirection;
direp:=Axis[ID].Ref.Status.PositiveDirection;
(*****************SysStep******************************)
CASE SysStep OF
0:	(*wait*)
	_00_Waiting();				
100:(*idle*)		
	_100_Idle();								
200:(*home*)		
	_200_Homing();
300:(*ready*)	
	_300_Ready();							
400:(*disable*)	
	_400_Disable();			
500:(*Moving*)
	_500_Moving();	
600:(*Stopping*)
	_600_Stopping();
700:(*Error*)
	_700_Error();	
800:(*Reset*)
	_800_Reset();		
END_CASE

(*****************Reset*************************)
IF GVL_API.stAxis[ID].reset OR GVL.Reset THEN 
	SysStep:=800;	
END_IF

ACT_SAFETY();


Axis[ID].aReadStatus();
Axis[ID].aReset();

ACTION _00_Waiting:
IF GVL_API.stAxis[ID].initialize THEN 
	GVL_API.stAxis[ID].initialize:=FALSE;
	Axis[ID].aStop(stop_do:=TRUE);
	SysStep:=100;
ELSIF GVL_API.stAxis[ID].homeExe THEN 
	GVL_API.stAxis[ID].homeExe:=FALSE;  
	GVL_API.stAxis[ID].Home_Done:=FALSE;
	SysStep:=200;
ELSIF GVL_API.stAxis[ID].MoveAbsoluteExe OR GVL_API.stAxis[ID].MoveRelativeExe 
		OR GVL_API.stAxis[ID].MoveVelocityExe OR GVL_API.stAxis[ID].JogBackwards 
		OR GVL_API.stAxis[ID].JogForward OR GVL_API.stAxis[ID].MoveConstantVelocity
		OR GVL_API.stAxis[ID].enabled OR GVL_API.stAxis[ID].Disable THEN 
	GVL_API.stAxis[ID].Move_Done:=FALSE;
	SysStep:=300;	
ELSIF GVL_API.stAxis[ID].stop THEN 
	SysStep:=600;	
ELSIF GVL_API.stAxis[ID].reset OR GVL.Reset THEN 
	SysStep:=800;	
END_IF

ton1(IN:=GVL_API.stAxis[ID].Home_Done OR  GVL_API.stAxis[ID].Move_Done , PT:=State_reset_time , Q=> , ET=> );
IF ton1.Q THEN 
	GVL_API.stAxis[ID].Home_Done:=FALSE;
	GVL_API.stAxis[ID].Move_Done:=FALSE;
END_IF
END_ACTION

ACTION _100_Idle:
Axis[ID].aStop(stop_do:=FALSE);
Axis[ID].aPower(power_do:=TRUE);	

IF axis[Id].Ref.Status .ControlLoopClosed THEN 
	GVL_API.stAxis[ID].state:=AxisStateEnum.idle;
	SysStep :=0;
ELSIF GVl.Emstop_Button OR GVL.Emstop_SAFE THEN 
	GVL_API.stAxis[ID].errorid:=Axis_XY_ErrorEnum.emergency_error;
	SysStep:=700;
END_IF

(*******************commandtimeout*********************************)
ton_commandtimeout(IN:=NOT axis[Id].Ref.Status .ControlLoopClosed , 
	PT:=LREAL_TO_TIME(GVL_API.stAxis[ID].commandtimeout*1000) ,
	Q=> , ET=> );
IF ton_commandtimeout.Q  THEN 
	ton_commandtimeout(IN:=FALSE );
	GVL_API.stAxis[ID].errorid:=Axis_XY_ErrorEnum.cmd_timeout;
	SysStep:=700;	
END_IF

(*****************RESET******************************)
IF GVL_API.stAxis[ID].reset OR GVL.HMI_btReset   THEN
	 SysStep:=800;
END_IF
END_ACTION

ACTION _200_Homing:
FB_Home(
		ref:=				Axis[ID].Ref , 
		Execute:= , 
		PosLimit:=			Axis[ID].IO.snLimitP , 
		Position:=			0 , 
		HomeingVelo:=		GVL_API.stAxis[ID].homingvelocity , 
		Standby_position:=  GVL_API.stAxis[ID].homeoffset,
		bCalibrationCam:=	Axis[ID].IO.snHome , 
		rel_dis:=			50 , 
		TimeOutSet:=		GVL_API.stAxis[ID].homingtimeout , 
		reset:= , 
		Done=> , 
		Busy=> , 
		Active=> , 
		CommandAborted=> , 
		Error=> , 
		ErrorID=> , 
		TimeOut=> );
		
CASE HomeStep OF
0:
	IF GVL_API.stAxis[ID].homingvelocity<>0 THEN 
		HomeStep:=10;
	END_IF
10:
	FB_Home.Execute:=TRUE;					
	IF FB_Home.Done THEN
		GVL_API.stAxis[ID].Home_Done:=TRUE;
		FB_Home.Execute:=FALSE;		
		HomeStep:=20;
	END_IF
	IF FB_Home.Error THEN 		
		GVL_API.stAxis[ID].ErrorId:=Axis_XY_ErrorEnum.homing_timeout;
		HomeStep:=30;
	END_IF
	
20:	(**********HOME DONE****************)	
	GVL_API.stAxis[ID].state:=AxisStateEnum.ready;	
	HomeStep:=0;	
	SysStep:=0;
		
30:(**********TIME OUT****************)
	FB_Home.Execute:=FALSE;
	FB_Home.reset:=TRUE;
	HomeStep:=40;
40:(**********RESET****************)
	FB_Home.reset:=FALSE;
	HomeStep:=0;
	SysStep:=700;
		
END_CASE

IF FB_Home.Busy THEN 
	GVL_API.stAxis[ID].state:=AxisStateEnum.homing;
END_IF


(*****************RESET******************************)
IF GVL_API.stAxis[ID].reset    THEN
	FB_Home.Execute:=FALSE;
	 SysStep:=800;
END_IF
END_ACTION

ACTION _300_Ready:
Axis[ID].aStop();
GVL_API.stAxis[ID].Move_Done:=FALSE;
(***********parameter_out_of_range***********)
IF GVL_API.stAxis[ID].requestedposition>GVL_API.stAxis[ID].maxDistance OR GVL_API.stAxis[ID].requestedposition<0 THEN 
		parameter_out_of_range:=TRUE;
ELSIF GVL_API.stAxis[ID].constantvelocitystart>GVL_API.stAxis[ID].maxDistance OR GVL_API.stAxis[ID].constantvelocitystart<0 THEN
		parameter_out_of_range:=TRUE;
ELSIF GVL_API.stAxis[ID].constanvelocityend>GVL_API.stAxis[ID].maxDistance OR GVL_API.stAxis[ID].constanvelocityend<0 THEN
		parameter_out_of_range:=TRUE;	
ELSIF  GVL_API.stAxis[ID].requestedoffset>0 
	AND (GVL_API.stAxis[ID].maxDistance-Axis[ID].Ref.NcToPlc.ActPos)<GVL_API.stAxis[ID].requestedoffset THEN
	 	parameter_out_of_range:=TRUE;
ELSIF GVL_API.stAxis[ID].requestedoffset<-1	
	AND Axis[ID].Ref.NcToPlc.ActPos<ABS(GVL_API.stAxis[ID].requestedoffset) THEN 
		parameter_out_of_range:=TRUE;

ELSE
		parameter_out_of_range:=FALSE;
END_IF	

(*********out_of_pos_range****************)
IF Axis[ID].Ref.NcToPlc.ActPos>GVL_API.stAxis[ID].maxDistance THEN 
	actuator_out_of_pos_range:=TRUE;
	actuator_out_of_neg_range:=FALSE;		
ELSIF	Axis[ID].Ref.NcToPlc.ActPos<-1 THEN 
	actuator_out_of_pos_range:=FALSE;
	actuator_out_of_neg_range:=TRUE;
ELSE
	actuator_out_of_pos_range:=FALSE;
	actuator_out_of_neg_range:=FALSE;
END_IF
	

(*****************state******************************)
IF Axis[ID].Ref.Status.NotMoving AND axis[Id].Ref.Status .ControlLoopClosed  
AND NOT Axis[ID].Ref.Status.Error THEN 
	IF parameter_out_of_range THEN 
		GVL_API.stAxis[ID].errorid:=Axis_XY_ErrorEnum.parameter_out_of_range;
		SysStep:=700;
	ELSIF actuator_out_of_pos_range THEN 
		GVL_API.stAxis[ID].errorid:=Axis_XY_ErrorEnum.actuator_out_of_pos_range;
		SysStep:=700;
	ELSIF actuator_out_of_neg_range THEN 
		GVL_API.stAxis[ID].errorid:=Axis_XY_ErrorEnum.actuator_out_of_neg_range;
		SysStep:=700;	
	ELSE
		GVL_API.stAxis[ID].state:=AxisStateEnum.ready;
		GVL_API.stAxis[ID].errorid:=Axis_XY_ErrorEnum.no_error;
	END_IF
END_IF

(*****************valid command******************************)
IF NOT parameter_out_of_range 
AND axis[Id].Ref.Status .ControlLoopClosed  THEN  			
	IF GVL_API.stAxis[ID].MoveAbsoluteExe OR GVL_API.stAxis[ID].MoveRelativeExe 
		OR GVL_API.stAxis[ID].MoveVelocityExe OR GVL_API.stAxis[ID].JogBackwards 
		OR GVL_API.stAxis[ID].JogForward OR GVL_API.stAxis[ID].MoveConstantVelocity	THEN 	  		
			SysStep:=500;		
	END_IF
END_IF

(*****************enable-disable******************************)
IF GVL_API.stAxis[ID].enabled THEN 
	Axis[Id].aPower(power_do:=TRUE);	
	GVL_API.stAxis[ID].enabled:=FALSE;
	 GVL_API.stAxis[ID].state:=AxisStateEnum.ready;
	SysStep :=0;
ELSIF  GVL_API.stAxis[ID].Disable THEN 
	  SysStep:=400;
END_IF


(*****************RESET******************************)
IF GVL_API.stAxis[ID].reset THEN
	 SysStep:=800;
END_IF
END_ACTION

ACTION _400_Disable:
(*****************enable-disable******************************)
IF GVL_API.stAxis[ID].Disable THEN 
	Axis[Id].aPower(power_do:=FALSE);
	GVL_API.stAxis[ID].Disable:=FALSE;
	GVL_API.stAxis[ID].state:=AxisStateEnum.disabled;
	//IF NOT  axis[Id].Ref.Status .ControlLoopClosed THEN 
		SysStep:=0;
	//END_IF
	
END_IF

(*****************RESET******************************)
IF GVL_API.stAxis[ID].reset THEN
	 SysStep:=800;
END_IF
END_ACTION

ACTION _500_Moving:
GVL_API.stAxis[ID].state:=AxisStateEnum.moving;

(*********out_of_pos_range****************)
IF Axis[ID].Ref.NcToPlc.ActPos>GVL_API.stAxis[ID].maxDistance THEN 
	actuator_out_of_pos_range:=TRUE;
	actuator_out_of_neg_range:=FALSE;
	GVL_API.stAxis[ID].JogForward:=FALSE;		
ELSIF	Axis[ID].Ref.NcToPlc.ActPos<-1 THEN 
	actuator_out_of_pos_range:=FALSE;
	actuator_out_of_neg_range:=TRUE;
	GVL_API.stAxis[ID].JogBackwards:=FALSE;
ELSE
	actuator_out_of_pos_range:=FALSE;
	actuator_out_of_neg_range:=FALSE;
END_IF

(*********parameter_out_of_range****************)
IF Axis[ID].IO.snHome 
	AND (GVL_API.stAxis[ID].requestedoffset<0 
	OR GVL_API.stAxis[ID].constantvelocitystart<Axis[ID].Ref.NcToPlc.ActPos
	OR GVL_API.stAxis[ID].constanvelocityend<Axis[ID].Ref.NcToPlc.ActPos
	OR GVL_API.stAxis[ID].requestedposition<Axis[ID].Ref.NcToPlc.ActPos)
	THEN 	parameter_out_of_range:=TRUE;
ELSIF Axis[ID].IO.snLimitP
	AND (GVL_API.stAxis[ID].requestedoffset>0 
	OR GVL_API.stAxis[ID].constantvelocitystart>Axis[ID].Ref.NcToPlc.ActPos
	OR GVL_API.stAxis[ID].constanvelocityend>Axis[ID].Ref.NcToPlc.ActPos
	OR GVL_API.stAxis[ID].requestedposition>Axis[ID].Ref.NcToPlc.ActPos)
	THEN 	parameter_out_of_range:=TRUE;
END_IF


IF NOT_Moving_TimeOut OR GVL_API.stAxis[ID].Move_Done  THEN 			(************NOT_Moving_TimeOut/Move_Done**************)
	NOT_Moving_TimeOut:=FALSE;	
	GVL_API.stAxis[ID].state:=AxisStateEnum.ready;			
	SysStep:=0;
ELSIF SpeedNotReach THEN 							(************SpeedNotReach**************)
	GVL_API.stAxis[ID].errorid:=Axis_XY_ErrorEnum.SpeedNotReach;
	SysStep:=700;
ELSIF Axis[ID].Ref.Status.NotMoving AND parameter_out_of_range THEN 
	GVL_API.stAxis[ID].errorid:=Axis_XY_ErrorEnum.parameter_out_of_range;
	SysStep:=700;
ELSIF Axis[ID].Ref.Status.Moving THEN 				(************trigger_limit**************)
	IF (Axis[ID].Ref.Status.NegativeDirection AND Axis[ID].IO.snLimitN) OR 
		(Axis[ID].Ref.Status.PositiveDirection AND Axis[ID].IO.snLimitP) 
		OR stInput.biElectromagnet_limit  OR stOutput.bqElectromagnet_power 
	THEN	
		Axis[ID].aStop(stop_do:=TRUE);
		GVL_API.stAxis[ID].errorid:=Axis_XY_ErrorEnum.trigger_limit;
		SysStep:=700;	
	END_IF 
	
ELSIF actuator_out_of_pos_range THEN 					(*********out_of_pos_range****************)
	Axis[ID].aStop(stop_do:=TRUE);
	GVL_API.stAxis[ID].errorid:=Axis_XY_ErrorEnum.actuator_out_of_pos_range;
	SysStep:=700;
ELSIF actuator_out_of_neg_range THEN
	Axis[ID].aStop(stop_do:=TRUE); 
	GVL_API.stAxis[ID].errorid:=Axis_XY_ErrorEnum.actuator_out_of_neg_range;
	SysStep:=700;	
ELSE GVL_API.stAxis[ID].errorid:=Axis_XY_ErrorEnum.no_error;
END_IF


(*****************JOG/ABS/REL/******************************)
(*****************MoveConstantVelocity*****************************)
IF NOT parameter_out_of_range  THEN 
	FB_move(
	enable:= 					NOT stInput.biElectromagnet_limit AND NOT stOutput.bqElectromagnet_power,	
	ref:= 						Axis[ID].Ref, 
	jogF:= 						GVL_API.stAxis[ID].JogForward, 
	jogB:= 						GVL_API.stAxis[ID].JogBackwards, 
	Move_Stop:=				GVL_API.stAxis[ID].stop OR GVL_API.stAxis[ID].reset ,
	PosLimit:=					Axis[ID].IO.snLimitP , 
	NegLimit:= 					Axis[ID].IO.snLimitN, 
	maxDistance:=				GVL_API.stAxis[ID].maxDistance ,	
	Acceleration:= 				GVL_API.stAxis[ID].acceleration, 
	Deceleration:= 				GVL_API.stAxis[ID].acceleration, 
	Jerk:= 						GVL_API.stAxis[ID].jerk, 	 
	MoveRelExe:= 				GVL_API.stAxis[ID].MoveRelativeExe, 
	MoveAbsExe:= 				GVL_API.stAxis[ID].MoveAbsoluteExe, 
	MoveConstantVelocityExe:= 	GVL_API.stAxis[ID].MoveConstantVelocity, 
	Velo:= 						GVL_API.stAxis[ID].velocity, 
	TargetRel:= 				GVL_API.stAxis[ID].requestedoffset, 
	TargetAbs:= 				GVL_API.stAxis[ID].requestedposition, 
	constantvelocitystart:= 	GVL_API.stAxis[ID].constantvelocitystart, 
	constanvelocityend:= 		GVL_API.stAxis[ID].constanvelocityend, 
	Done:= 						GVL_API.stAxis[ID].Move_Done,
	NotMovingTimeOut:= 			NOT_Moving_TimeOut,
	SpeedNotReach:=				SpeedNotReach
	);	
END_IF


(*****************stop******************************)
IF GVL_API.stAxis[ID].stop THEN 
	SysStep:=600;
END_IF
(*****************RESET******************************)
IF GVL_API.stAxis[ID].reset THEN
	 SysStep:=800;
END_IF
END_ACTION

ACTION _600_Stopping:
(**************只单独用作STOP命令*************************)
GVL_API.stAxis[ID].state:=AxisStateEnum.stopping;

Axis[ID].aStop(stop_do:=GVL_API.stAxis[ID].stop,Jerk:=GVL_API.stAxis[ID].jerk);
IF Axis[ID].mcStop.Busy THEN 
	GVL_API.stAxis[ID].state:=AxisStateEnum.stopping;	
	GVL_API.stAxis[ID].JogBackwards:=FALSE;
	GVL_API.stAxis[ID].JogForward:=FALSE;
	GVL_API.stAxis[ID].MoveAbsoluteExe:=FALSE;
	GVL_API.stAxis[ID].MoveConstantVelocity:=FALSE;
	GVL_API.stAxis[ID].MoveRelativeExe:=FALSE;
	GVL_API.stAxis[ID].velocity:=0;
	GVL_API.stAxis[ID].requestedoffset:=0;
	GVL_API.stAxis[ID].requestedposition:=0;
	GVL_API.stAxis[ID].stop:=FALSE;
END_IF

IF Axis[ID].mcStop.Done AND Axis[ID].Ref.Status.NotMoving   THEN 		
	GVL_API.stAxis[ID].stop:=FALSE;
	GVL_API.stAxis[ID].state:=AxisStateEnum.ready;	
	GVL_API.stAxis[ID].Move_Done:=TRUE;
	SysStep:=0;
END_IF

(*****************RESET******************************)
IF GVL_API.stAxis[ID].reset THEN
	 GVL_API.stAxis[ID].stop:=FALSE;
	 Axis[ID].aStop(stop_do:=FALSE);
	 SysStep:=800;
END_IF
END_ACTION

ACTION _700_Error:
(*****************ERROR******************************)
GVL_API.stAxis[ID].Error:=TRUE;
GVL_API.stAxis[ID].state:=AxisStateEnum.error;
		GVL_API.stAxis[ID].initialize:=FALSE;
		GVL_API.stAxis[ID].homeExe:=FALSE; 
		GVL_API.stAxis[ID].stop:=FALSE;
		GVL_API.stAxis[ID].JogBackwards:=FALSE;
		GVL_API.stAxis[ID].JogForward:=FALSE;
		GVL_API.stAxis[ID].MoveAbsoluteExe:=FALSE;
		GVL_API.stAxis[ID].MoveConstantVelocity:=FALSE;
		GVL_API.stAxis[ID].MoveRelativeExe:=FALSE;
		GVL_API.stAxis[ID].velocity:=0;
		GVL_API.stAxis[ID].requestedoffset:=0;
		GVL_API.stAxis[ID].requestedposition:=0;
		GVL_API.stAxis[ID].constantvelocitystart:=0;
		GVL_API.stAxis[ID].constanvelocityend:=0;
		FB_Home.Execute:=FALSE;
		GVL_API.stAxis[ID].Home_Done:=FALSE;
		GVL_API.stAxis[ID].Move_Done:=FALSE;
 SysStep:=0;
END_ACTION

